LIN {X 0,Y 404.373,Z 885.046,A -85,B 0,C 180,E1 -11042.423,E2 -11042.423} C_VEL
LIN {X 0,Y 404.228,Z 886.16,A -85,B 0,C 180,E1 -11044.238,E2 -11044.238} C_VEL
LIN {X 0,Y 404.158,Z 886.18,A -85,B 0,C 180,E1 -11045.335,E2 -11045.335} C_VEL
LIN {X 0,Y 404.188,Z 885.21,A -85,B 0,C 180,E1 -11047.156,E2 -11047.156} C_VEL
LIN {X 0,Y 404.359,Z 883.5,A -85,B 0,C 180,E1 -11048.595,E2 -11048.595} C_VEL
LIN {X 0,Y 404.64,Z 880.506,A -85,B 0,C 180,E1 -11050.237,E2 -11050.237} C_VEL
LIN {X 0,Y 404.956,Z 876.549,A -85,B 0,C 180,E1 -11051.798,E2 -11051.798} C_VEL
LIN {X 0,Y 405.434,Z 871.294,A -85,B 0,C 180,E1 -11053.382,E2 -11053.382} C_VEL
LIN {X 0,Y 405.955,Z 864.651,A -85,B 0,C 180,E1 -11054.95,E2 -11054.95} C_VEL
LIN {X 0,Y 406.678,Z 856.301,A -85,B 0,C 180,E1 -11056.51,E2 -11056.51} C_VEL
LIN {X 0,Y 407.287,Z 847.808,A -85,B 0,C 180,E1 -11057.798,E2 -11057.798} C_VEL
LIN {X 0,Y 407.94,Z 838.484,A -85,B 0,C 180,E1 -11058.952,E2 -11058.952} C_VEL
LIN {X 0,Y 408.542,Z 828.149,A -85,B 0,C 180,E1 -11059.986,E2 -11059.986} C_VEL
LIN {X 0,Y 409.118,Z 817.223,A -85,B 0,C 180,E1 -11060.858,E2 -11060.858} C_VEL
LIN {X 0,Y 409.51,Z 805.087,A -85,B 0,C 180,E1 -11061.613,E2 -11061.613} C_VEL
LIN {X 0,Y 409.764,Z 792.492,A -85,B 0,C 180,E1 -11062.177,E2 -11062.177} C_VEL
LIN {X 0,Y 409.872,Z 779.499,A -85,B 0,C 180,E1 -11062.551,E2 -11062.551} C_VEL
LIN {X 0,Y 410.43,Z 724.572,A -85,B 0,C 180,E1 -11063.541,E2 -11063.541} C_VEL
LIN {X 0,Y 409.821,Z 721.492,A -85,B 0,C 180,E1 -11063.627,E2 -11063.627} C_VEL
LIN {X 0,Y 407.436,Z 717.769,A -85,B 0,C 180,E1 -11063.81,E2 -11063.81} C_VEL
LIN {X 0,Y 401.011,Z 711.142,A -85,B 0,C 180,E1 -11064.25,E2 -11064.25} C_VEL
LIN {X 0,Y 399.002,Z 707.692,A -85,B 0,C 180,E1 -11064.415,E2 -11064.415} C_VEL
LIN {X 0,Y 397.415,Z 703.698,A -85,B 0,C 180,E1 -11064.614,E2 -11064.614} C_VEL
LIN {X 0,Y 397.262,Z 703.081,A -85,B 0,C 180,E1 -11064.787,E2 -11064.787} C_VEL
LIN {X 0,Y 397.442,Z 702.978,A -85,B 0,C 180,E1 -11067.975,E2 -11067.975} C_VEL
LIN {X 0,Y 397.441,Z 702.977,A -85,B 0,C 180,E1 -11072.028,E2 -11072.028} C_VEL
LIN {X 0,Y 397.324,Z 702.996,A -85,B 0,C 180,E1 -11076.094,E2 -11076.094} C_VEL
LIN {X 0,Y 397.23,Z 703.003,A -85,B 0,C 180,E1 -11079.164,E2 -11079.164} C_VEL
LIN {X 0,Y 397.218,Z 703.004,A -85,B 0,C 180,E1 -11082.26,E2 -11082.26} C_VEL
LIN {X 0,Y 397.178,Z 703.005,A -85,B 0,C 180,E1 -11085.393,E2 -11085.393} C_VEL
LIN {X 0,Y 397.146,Z 703.013,A -85,B 0,C 180,E1 -11088.576,E2 -11088.576} C_VEL
LIN {X 0,Y 397.098,Z 703.016,A -85,B 0,C 180,E1 -11091.82,E2 -11091.82} C_VEL
LIN {X 0,Y 397.107,Z 703.011,A -85,B 0,C 180,E1 -11095.136,E2 -11095.136} C_VEL
LIN {X 0,Y 397.066,Z 703.017,A -85,B 0,C 180,E1 -11098.55,E2 -11098.55} C_VEL
LIN {X 0,Y 397.081,Z 703.017,A -85,B 0,C 180,E1 -11101.835,E2 -11101.835} C_VEL
LIN {X 0,Y 397.121,Z 702.997,A -85,B 0,C 180,E1 -11104.495,E2 -11104.495} C_VEL
LIN {X 0,Y 397.092,Z 703.016,A -85,B 0,C 180,E1 -11108.278,E2 -11108.278} C_VEL
LIN {X 0,Y 397.051,Z 703.024,A -85,B 0,C 180,E1 -11110.915,E2 -11110.915} C_VEL
LIN {X 0,Y 397.083,Z 703.02,A -85,B 0,C 180,E1 -11114.93,E2 -11114.93} C_VEL
LIN {X 0,Y 397.057,Z 703.026,A -85,B 0,C 180,E1 -11118.024,E2 -11118.024} C_VEL
LIN {X 0,Y 397.093,Z 703.02,A -85,B 0,C 180,E1 -11121.147,E2 -11121.147} C_VEL
LIN {X 0,Y 397.096,Z 703.021,A -85,B 0,C 180,E1 -11124.503,E2 -11124.503} C_VEL
LIN {X 0,Y 397.119,Z 703.2,A -85,B 0,C 180,E1 -11127.857,E2 -11127.857} C_VEL
LIN {X 0,Y 397.298,Z 704.02,A -85,B 0,C 180,E1 -11128.009,E2 -11128.009} C_VEL
LIN {X 0,Y 402.683,Z 719.124,A -85,B 0,C 180,E1 -11128.58,E2 -11128.58} C_VEL
LIN {X 0,Y 401.817,Z 779.52,A -85,B 0,C 180,E1 -11129.829,E2 -11129.829} C_VEL
LIN {X 0,Y 401.599,Z 791.294,A -85,B 0,C 180,E1 -11130.227,E2 -11130.227} C_VEL
LIN {X 0,Y 401.342,Z 801.779,A -85,B 0,C 180,E1 -11130.724,E2 -11130.724} C_VEL
LIN {X 0,Y 401.038,Z 811.202,A -85,B 0,C 180,E1 -11131.293,E2 -11131.293} C_VEL
LIN {X 0,Y 400.595,Z 820.808,A -85,B 0,C 180,E1 -11132.011,E2 -11132.011} C_VEL
LIN {X 0,Y 400.075,Z 831.074,A -85,B 0,C 180,E1 -11132.962,E2 -11132.962} C_VEL
LIN {X 0,Y 399.546,Z 839.6,A -85,B 0,C 180,E1 -11133.912,E2 -11133.912} C_VEL
LIN {X 0,Y 399.101,Z 847.754,A -85,B 0,C 180,E1 -11134.999,E2 -11134.999} C_VEL
LIN {X 0,Y 398.681,Z 854.642,A -85,B 0,C 180,E1 -11136.081,E2 -11136.081} C_VEL
LIN {X 0,Y 398.145,Z 861.775,A -85,B 0,C 180,E1 -11137.422,E2 -11137.422} C_VEL
LIN {X 0,Y 397.75,Z 867.648,A -85,B 0,C 180,E1 -11138.763,E2 -11138.763} C_VEL
LIN {X 0,Y 397.539,Z 871.976,A -85,B 0,C 180,E1 -11139.945,E2 -11139.945} C_VEL
LIN {X 0,Y 397.261,Z 876.335,A -85,B 0,C 180,E1 -11141.431,E2 -11141.431} C_VEL
LIN {X 0,Y 397.098,Z 879.609,A -85,B 0,C 180,E1 -11142.888,E2 -11142.888} C_VEL
LIN {X 0,Y 396.942,Z 882.245,A -85,B 0,C 180,E1 -11144.598,E2 -11144.598} C_VEL
LIN {X 0,Y 396.906,Z 883.373,A -85,B 0,C 180,E1 -11145.647,E2 -11145.647} C_VEL
LIN {X 0,Y 396.939,Z 883.999,A -85,B 0,C 180,E1 -11146.861,E2 -11146.861} C_VEL
LIN {X 0,Y 397.061,Z 883.862,A -85,B 0,C 180,E1 -11148.773,E2 -11148.773} C_VEL
LIN {X 0,Y 397.327,Z 881.934,A -85,B 0,C 180,E1 -11150.84,E2 -11150.84} C_VEL
LIN {X 0,Y 397.605,Z 879.747,A -85,B 0,C 180,E1 -11152.211,E2 -11152.211} C_VEL
LIN {X 0,Y 397.873,Z 877.209,A -85,B 0,C 180,E1 -11153.407,E2 -11153.407} C_VEL
LIN {X 0,Y 398.275,Z 872.869,A -85,B 0,C 180,E1 -11154.938,E2 -11154.938} C_VEL
LIN {X 0,Y 398.75,Z 867.283,A -85,B 0,C 180,E1 -11156.463,E2 -11156.463} C_VEL
LIN {X 0,Y 399.295,Z 861.568,A -85,B 0,C 180,E1 -11157.73,E2 -11157.73} C_VEL
LIN {X 0,Y 399.927,Z 854.651,A -85,B 0,C 180,E1 -11158.993,E2 -11158.993} C_VEL
LIN {X 0,Y 400.608,Z 846.07,A -85,B 0,C 180,E1 -11160.276,E2 -11160.276} C_VEL
LIN {X 0,Y 401.152,Z 838.689,A -85,B 0,C 180,E1 -11161.2,E2 -11161.2} C_VEL
LIN {X 0,Y 401.806,Z 829.752,A -85,B 0,C 180,E1 -11162.13,E2 -11162.13} C_VEL
LIN {X 0,Y 402.229,Z 821.185,A -85,B 0,C 180,E1 -11162.879,E2 -11162.879} C_VEL
LIN {X 0,Y 402.653,Z 810.512,A -85,B 0,C 180,E1 -11163.627,E2 -11163.627} C_VEL
LIN {X 0,Y 403.032,Z 800.219,A -85,B 0,C 180,E1 -11164.187,E2 -11164.187} C_VEL
LIN {X 0,Y 403.228,Z 789.583,A -85,B 0,C 180,E1 -11164.624,E2 -11164.624} C_VEL
LIN {X 0,Y 403.267,Z 777.527,A -85,B 0,C 180,E1 -11164.968,E2 -11164.968} C_VEL
LIN {X 0,Y 404.446,Z 720.258,A -85,B 0,C 180,E1 -11166.218,E2 -11166.218} C_VEL
LIN {X 0,Y 399.902,Z 709.007,A -85,B 0,C 180,E1 -11166.793,E2 -11166.793} C_VEL
LIN {X 0,Y 397.46,Z 703.744,A -85,B 0,C 180,E1 -11167.138,E2 -11167.138} C_VEL
LIN {X 0,Y 397.343,Z 703.058,A -85,B 0,C 180,E1 -11167.339,E2 -11167.339} C_VEL
LIN {X 0,Y 397.205,Z 703.008,A -85,B 0,C 180,E1 -11171.223,E2 -11171.223} C_VEL
LIN {X 0,Y 397.184,Z 703.011,A -85,B 0,C 180,E1 -11174.343,E2 -11174.343} C_VEL
LIN {X 0,Y 397.152,Z 703.013,A -85,B 0,C 180,E1 -11177.508,E2 -11177.508} C_VEL
LIN {X 0,Y 397.11,Z 703.021,A -85,B 0,C 180,E1 -11180.729,E2 -11180.729} C_VEL
LIN {X 0,Y 397.131,Z 703.015,A -85,B 0,C 180,E1 -11184.018,E2 -11184.018} C_VEL
LIN {X 0,Y 397.122,Z 703.017,A -85,B 0,C 180,E1 -11187.763,E2 -11187.763} C_VEL
LIN {X 0,Y 397.085,Z 703.023,A -85,B 0,C 180,E1 -11190.882,E2 -11190.882} C_VEL
LIN {X 0,Y 397.131,Z 703.015,A -85,B 0,C 180,E1 -11194.493,E2 -11194.493} C_VEL
LIN {X 0,Y 397.11,Z 703.018,A -85,B 0,C 180,E1 -11198.274,E2 -11198.274} C_VEL
LIN {X 0,Y 397.095,Z 703.021,A -85,B 0,C 180,E1 -11200.908,E2 -11200.908} C_VEL
LIN {X 0,Y 397.108,Z 703.021,A -85,B 0,C 180,E1 -11203.648,E2 -11203.648} C_VEL
LIN {X 0,Y 397.108,Z 703.018,A -85,B 0,C 180,E1 -11206.52,E2 -11206.52} C_VEL
LIN {X 0,Y 397.118,Z 703.016,A -85,B 0,C 180,E1 -11210.422,E2 -11210.422} C_VEL
LIN {X 0,Y 397.113,Z 703.018,A -85,B 0,C 180,E1 -11214.264,E2 -11214.264} C_VEL
LIN {X 0,Y 397.152,Z 703.193,A -85,B 0,C 180,E1 -11216.375,E2 -11216.375} C_VEL
LIN {X 0,Y 401.047,Z 719.548,A -85,B 0,C 180,E1 -11219.455,E2 -11219.455} C_VEL
LIN {X 0,Y 402.871,Z 729.169,A -85,B 0,C 180,E1 -11221.156,E2 -11221.156} C_VEL
LIN {X 0,Y 400.963,Z 752.371,A -85,B 0,C 180,E1 -11224.845,E2 -11224.845} C_VEL
LIN {X 0,Y 399.627,Z 772.769,A -85,B 0,C 180,E1 -11228.054,E2 -11228.054} C_VEL
LIN {X 0,Y 398.971,Z 784.14,A -85,B 0,C 180,E1 -11229.808,E2 -11229.808} C_VEL
LIN {X 0,Y 400.351,Z 797.906,A -85,B 0,C 180,E1 -11230.261,E2 -11230.261} C_VEL
LIN {X 0,Y 403.016,Z 825.383,A -85,B 0,C 180,E1 -11230.899,E2 -11230.899} C_VEL
LIN {X 0,Y 402.062,Z 895.502,A -85,B 0,C 180,E1 -11232.186,E2 -11232.186} C_VEL
LIN {X 0,Y 401.522,Z 908.77,A -85,B 0,C 180,E1 -11232.622,E2 -11232.622} C_VEL
LIN {X 0,Y 400.721,Z 921.535,A -85,B 0,C 180,E1 -11233.243,E2 -11233.243} C_VEL
LIN {X 0,Y 399.835,Z 933.73,A -85,B 0,C 180,E1 -11234.058,E2 -11234.058} C_VEL
LIN {X 0,Y 398.861,Z 945.354,A -85,B 0,C 180,E1 -11235.065,E2 -11235.065} C_VEL
LIN {X 0,Y 398.127,Z 955.313,A -85,B 0,C 180,E1 -11236.144,E2 -11236.144} C_VEL
LIN {X 0,Y 397.63,Z 963.618,A -85,B 0,C 180,E1 -11237.235,E2 -11237.235} C_VEL
LIN {X 0,Y 397.003,Z 971.74,A -85,B 0,C 180,E1 -11238.511,E2 -11238.511} C_VEL
LIN {X 0,Y 396.572,Z 979.734,A -85,B 0,C 180,E1 -11240.049,E2 -11240.049} C_VEL
LIN {X 0,Y 396.359,Z 987.083,A -85,B 0,C 180,E1 -11241.844,E2 -11241.844} C_VEL
LIN {X 0,Y 396.291,Z 991.709,A -85,B 0,C 180,E1 -11243.281,E2 -11243.281} C_VEL
LIN {X 0,Y 396.396,Z 995.766,A -85,B 0,C 180,E1 -11244.913,E2 -11244.913} C_VEL
LIN {X 0,Y 396.519,Z 997.717,A -85,B 0,C 180,E1 -11245.933,E2 -11245.933} C_VEL
LIN {X 0,Y 396.457,Z 999.165,A -85,B 0,C 180,E1 -11246.95,E2 -11246.95} C_VEL
LIN {X 0,Y 396.478,Z 1000.191,A -85,B 0,C 180,E1 -11247.967,E2 -11247.967} C_VEL
LIN {X 0,Y 396.511,Z 1000.812,A -85,B 0,C 180,E1 -11248.983,E2 -11248.983} C_VEL
LIN {X 0,Y 396.541,Z 1001.028,A -85,B 0,C 180,E1 -11249.998,E2 -11249.998} C_VEL
LIN {X 0,Y 396.513,Z 1000.791,A -85,B 0,C 180,E1 -11251.014,E2 -11251.014} C_VEL
LIN {X 0,Y 396.483,Z 1000.134,A -85,B 0,C 180,E1 -11252.03,E2 -11252.03} C_VEL
LIN {X 0,Y 396.461,Z 999.074,A -85,B 0,C 180,E1 -11253.047,E2 -11253.047} C_VEL
LIN {X 0,Y 396.504,Z 997.609,A -85,B 0,C 180,E1 -11254.064,E2 -11254.064} C_VEL
LIN {X 0,Y 396.319,Z 994.499,A -85,B 0,C 180,E1 -11255.596,E2 -11255.596} C_VEL
LIN {X 0,Y 396.307,Z 990.341,A -85,B 0,C 180,E1 -11257.129,E2 -11257.129} C_VEL
LIN {X 0,Y 396.413,Z 983.991,A -85,B 0,C 180,E1 -11258.923,E2 -11258.923} C_VEL
LIN {X 0,Y 396.648,Z 977.08,A -85,B 0,C 180,E1 -11260.462,E2 -11260.462} C_VEL
LIN {X 0,Y 397.159,Z 968.562,A -85,B 0,C 180,E1 -11261.999,E2 -11261.999} C_VEL
LIN {X 0,Y 397.892,Z 959.904,A -85,B 0,C 180,E1 -11263.273,E2 -11263.273} C_VEL
LIN {X 0,Y 398.548,Z 950.429,A -85,B 0,C 180,E1 -11264.421,E2 -11264.421} C_VEL
LIN {X 0,Y 399.276,Z 940.172,A -85,B 0,C 180,E1 -11265.438,E2 -11265.438} C_VEL
LIN {X 0,Y 400.222,Z 929.079,A -85,B 0,C 180,E1 -11266.316,E2 -11266.316} C_VEL
LIN {X 0,Y 401.113,Z 916.855,A -85,B 0,C 180,E1 -11267.065,E2 -11267.065} C_VEL
LIN {X 0,Y 401.862,Z 904.313,A -85,B 0,C 180,E1 -11267.622,E2 -11267.622} C_VEL
LIN {X 0,Y 402.353,Z 891.365,A -85,B 0,C 180,E1 -11267.994,E2 -11267.994} C_VEL
LIN {X 0,Y 403.171,Z 822.843,A -85,B 0,C 180,E1 -11269.249,E2 -11269.249} C_VEL
LIN {X 0,Y 399.24,Z 786.031,A -85,B 0,C 180,E1 -11270.158,E2 -11270.158} C_VEL
LIN {X 0,Y 398.849,Z 782.941,A -85,B 0,C 180,E1 -11270.263,E2 -11270.263} C_VEL
LIN {X 0,Y 400.24,Z 761.86,A -85,B 0,C 180,E1 -11273.544,E2 -11273.544} C_VEL
LIN {X 0,Y 402.273,Z 734.827,A -85,B 0,C 180,E1 -11277.86,E2 -11277.86} C_VEL
LIN {X 0,Y 402.746,Z 727.843,A -85,B 0,C 180,E1 -11278.999,E2 -11278.999} C_VEL
LIN {X 0,Y 400.176,Z 715.833,A -85,B 0,C 180,E1 -11281.201,E2 -11281.201} C_VEL
LIN {X 0,Y 397.136,Z 703.138,A -85,B 0,C 180,E1 -11283.696,E2 -11283.696} C_VEL
LIN {X 0,Y 397.087,Z 703.023,A -85,B 0,C 180,E1 -11287.207,E2 -11287.207} C_VEL
LIN {X 0,Y 397.094,Z 703.019,A -85,B 0,C 180,E1 -11290.444,E2 -11290.444} C_VEL
LIN {X 0,Y 397.093,Z 703.018,A -85,B 0,C 180,E1 -11293.647,E2 -11293.647} C_VEL
LIN {X 0,Y 397.097,Z 703.015,A -85,B 0,C 180,E1 -11296.519,E2 -11296.519} C_VEL
LIN {X 0,Y 397.105,Z 703.009,A -85,B 0,C 180,E1 -11300.422,E2 -11300.422} C_VEL
LIN {X 0,Y 397.099,Z 703.01,A -85,B 0,C 180,E1 -11304.264,E2 -11304.264} C_VEL
LIN {X 0,Y 397.104,Z 703.018,A -85,B 0,C 180,E1 -11306.726,E2 -11306.726} C_VEL
LIN {X 0,Y 397.123,Z 703.016,A -85,B 0,C 180,E1 -11310.296,E2 -11310.296} C_VEL
LIN {X 0,Y 397.184,Z 703.006,A -85,B 0,C 180,E1 -11312.609,E2 -11312.609} C_VEL
LIN {X 0,Y 397.122,Z 703.017,A -85,B 0,C 180,E1 -11315.981,E2 -11315.981} C_VEL
LIN {X 0,Y 397.127,Z 703.016,A -85,B 0,C 180,E1 -11319.704,E2 -11319.704} C_VEL
LIN {X 0,Y 397.172,Z 703.002,A -85,B 0,C 180,E1 -11322.843,E2 -11322.843} C_VEL
LIN {X 0,Y 397.166,Z 703.012,A -85,B 0,C 180,E1 -11325.657,E2 -11325.657} C_VEL
LIN {X 0,Y 397.187,Z 703.007,A -85,B 0,C 180,E1 -11328.776,E2 -11328.776} C_VEL
LIN {X 0,Y 397.349,Z 702.985,A -85,B 0,C 180,E1 -11332.076,E2 -11332.076} C_VEL
LIN {X 0,Y 397.243,Z 702.996,A -85,B 0,C 180,E1 -11334.925,E2 -11334.925} C_VEL
LIN {X 0,Y 397.44,Z 702.977,A -85,B 0,C 180,E1 -11337.973,E2 -11337.973} C_VEL
LIN {X 0,Y 397.568,Z 702.957,A -85,B 0,C 180,E1 -11340,E2 -11340} C_VEL
LIN {X 0,Y 397.369,Z 702.983,A -85,B 0,C 180,E1 -11343.042,E2 -11343.042} C_VEL
LIN {X 0,Y 397.35,Z 702.987,A -85,B 0,C 180,E1 -11347.112,E2 -11347.112} C_VEL
LIN {X 0,Y 397.207,Z 703.005,A -85,B 0,C 180,E1 -11350.192,E2 -11350.192} C_VEL
LIN {X 0,Y 397.215,Z 703.005,A -85,B 0,C 180,E1 -11353.322,E2 -11353.322} C_VEL
LIN {X 0,Y 397.17,Z 703.014,A -85,B 0,C 180,E1 -11357.156,E2 -11357.156} C_VEL
LIN {X 0,Y 397.091,Z 703.021,A -85,B 0,C 180,E1 -11360.731,E2 -11360.731} C_VEL
LIN {X 0,Y 397.114,Z 703.006,A -85,B 0,C 180,E1 -11364.02,E2 -11364.02} C_VEL
LIN {X 0,Y 397.184,Z 703.006,A -85,B 0,C 180,E1 -11367.391,E2 -11367.391} C_VEL
LIN {X 0,Y 397.069,Z 703.026,A -85,B 0,C 180,E1 -11370.884,E2 -11370.884} C_VEL
LIN {X 0,Y 397.117,Z 703.017,A -85,B 0,C 180,E1 -11374.495,E2 -11374.495} C_VEL
LIN {X 0,Y 397.099,Z 703.016,A -85,B 0,C 180,E1 -11378.276,E2 -11378.276} C_VEL
LIN {X 0,Y 397.082,Z 703.02,A -85,B 0,C 180,E1 -11380.91,E2 -11380.91} C_VEL
LIN {X 0,Y 397.094,Z 703.022,A -85,B 0,C 180,E1 -11383.65,E2 -11383.65} C_VEL
LIN {X 0,Y 397.133,Z 703.284,A -85,B 0,C 180,E1 -11385.063,E2 -11385.063} C_VEL
LIN {X 0,Y 397.457,Z 704.485,A -85,B 0,C 180,E1 -11385.222,E2 -11385.222} C_VEL
LIN {X 0,Y 404.151,Z 720.562,A -85,B 0,C 180,E1 -11385.923,E2 -11385.923} C_VEL
LIN {X 0,Y 403.609,Z 785.345,A -85,B 0,C 180,E1 -11387.147,E2 -11387.147} C_VEL
LIN {X 0,Y 403.48,Z 798.403,A -85,B 0,C 180,E1 -11387.593,E2 -11387.593} C_VEL
LIN {X 0,Y 403.24,Z 810.296,A -85,B 0,C 180,E1 -11388.193,E2 -11388.193} C_VEL
LIN {X 0,Y 402.814,Z 821.878,A -85,B 0,C 180,E1 -11388.972,E2 -11388.972} C_VEL
LIN {X 0,Y 402.139,Z 832.712,A -85,B 0,C 180,E1 -11389.906,E2 -11389.906} C_VEL
LIN {X 0,Y 401.408,Z 843.546,A -85,B 0,C 180,E1 -11391.091,E2 -11391.091} C_VEL
LIN {X 0,Y 400.549,Z 853.417,A -85,B 0,C 180,E1 -11392.433,E2 -11392.433} C_VEL
LIN {X 0,Y 399.847,Z 861.013,A -85,B 0,C 180,E1 -11393.711,E2 -11393.711} C_VEL
LIN {X 0,Y 399.259,Z 867.779,A -85,B 0,C 180,E1 -11395.106,E2 -11395.106} C_VEL
LIN {X 0,Y 398.531,Z 874.56,A -85,B 0,C 180,E1 -11396.863,E2 -11396.863} C_VEL
LIN {X 0,Y 397.997,Z 879.692,A -85,B 0,C 180,E1 -11398.608,E2 -11398.608} C_VEL
LIN {X 0,Y 397.636,Z 883.349,A -85,B 0,C 180,E1 -11400.34,E2 -11400.34} C_VEL
LIN {X 0,Y 397.368,Z 885.865,A -85,B 0,C 180,E1 -11402.169,E2 -11402.169} C_VEL
LIN {X 0,Y 397.22,Z 886.998,A -85,B 0,C 180,E1 -11403.75,E2 -11403.75} C_VEL
LIN {X 0,Y 397.17,Z 887.244,A -85,B 0,C 180,E1 -11404.871,E2 -11404.871} C_VEL
LIN {X 0,Y 397.122,Z 887.004,A -85,B 0,C 180,E1 -11405.983,E2 -11405.983} C_VEL
LIN {X 0,Y 397.176,Z 886.288,A -85,B 0,C 180,E1 -11407.092,E2 -11407.092} C_VEL
LIN {X 0,Y 397.304,Z 885.138,A -85,B 0,C 180,E1 -11408.195,E2 -11408.195} C_VEL
LIN {X 0,Y 397.516,Z 883.004,A -85,B 0,C 180,E1 -11409.56,E2 -11409.56} C_VEL
LIN {X 0,Y 397.886,Z 878.772,A -85,B 0,C 180,E1 -11411.463,E2 -11411.463} C_VEL
LIN {X 0,Y 398.337,Z 873.834,A -85,B 0,C 180,E1 -11413.077,E2 -11413.077} C_VEL
LIN {X 0,Y 398.884,Z 867.576,A -85,B 0,C 180,E1 -11414.677,E2 -11414.677} C_VEL
LIN {X 0,Y 399.547,Z 859.778,A -85,B 0,C 180,E1 -11416.265,E2 -11416.265} C_VEL
LIN {X 0,Y 400.195,Z 851.76,A -85,B 0,C 180,E1 -11417.579,E2 -11417.579} C_VEL
LIN {X 0,Y 400.905,Z 841.957,A -85,B 0,C 180,E1 -11418.883,E2 -11418.883} C_VEL
LIN {X 0,Y 401.613,Z 831.064,A -85,B 0,C 180,E1 -11420.051,E2 -11420.051} C_VEL
LIN {X 0,Y 402.227,Z 820.431,A -85,B 0,C 180,E1 -11420.954,E2 -11420.954} C_VEL
LIN {X 0,Y 402.718,Z 807.73,A -85,B 0,C 180,E1 -11421.787,E2 -11421.787} C_VEL
LIN {X 0,Y 403.012,Z 795.141,A -85,B 0,C 180,E1 -11422.392,E2 -11422.392} C_VEL
LIN {X 0,Y 403.092,Z 782.076,A -85,B 0,C 180,E1 -11422.803,E2 -11422.803} C_VEL
LIN {X 0,Y 403.757,Z 720.112,A -85,B 0,C 180,E1 -11423.944,E2 -11423.944} C_VEL
LIN {X 0,Y 399.002,Z 707.692,A -85,B 0,C 180,E1 -11424.415,E2 -11424.415} C_VEL
LIN {X 0,Y 397.975,Z 705.732,A -85,B 0,C 180,E1 -11424.588,E2 -11424.588} C_VEL
LIN {X 0,Y 396.428,Z 704.172,A -85,B 0,C 180,E1 -11424.976,E2 -11424.976} C_VEL
LIN {X 0,Y 394.554,Z 703.476,A -85,B 0,C 180,E1 -11425.595,E2 -11425.595} C_VEL
LIN {X 0,Y 392.119,Z 703.641,A -85,B 0,C 180,E1 -11426.765,E2 -11426.765} C_VEL
LIN {X 0,Y 390.564,Z 703.835,A -85,B 0,C 180,E1 -11428.074,E2 -11428.074} C_VEL
LIN {X 0,Y 390.307,Z 703.866,A -85,B 0,C 180,E1 -11428.738,E2 -11428.738} C_VEL
LIN {X 0,Y 390.407,Z 703.853,A -85,B 0,C 180,E1 -11432.065,E2 -11432.065} C_VEL
LIN {X 0,Y 390.28,Z 703.873,A -85,B 0,C 180,E1 -11436.204,E2 -11436.204} C_VEL
LIN {X 0,Y 390.189,Z 703.879,A -85,B 0,C 180,E1 -11439.331,E2 -11439.331} C_VEL
LIN {X 0,Y 390.201,Z 703.876,A -85,B 0,C 180,E1 -11443.44,E2 -11443.44} C_VEL
LIN {X 0,Y 390.135,Z 703.887,A -85,B 0,C 180,E1 -11447.299,E2 -11447.299} C_VEL
LIN {X 0,Y 390.056,Z 703.892,A -85,B 0,C 180,E1 -11451.124,E2 -11451.124} C_VEL
LIN {X 0,Y 390.048,Z 703.897,A -85,B 0,C 180,E1 -11454.484,E2 -11454.484} C_VEL
LIN {X 0,Y 390.022,Z 703.893,A -85,B 0,C 180,E1 -11457.998,E2 -11457.998} C_VEL
LIN {X 0,Y 390.023,Z 703.899,A -85,B 0,C 180,E1 -11461.506,E2 -11461.506} C_VEL
LIN {X 0,Y 390.073,Z 703.874,A -85,B 0,C 180,E1 -11465.21,E2 -11465.21} C_VEL
LIN {X 0,Y 390.06,Z 703.895,A -85,B 0,C 180,E1 -11469.098,E2 -11469.098} C_VEL
LIN {X 0,Y 390.014,Z 703.9,A -85,B 0,C 180,E1 -11472.369,E2 -11472.369} C_VEL
LIN {X 0,Y 390.049,Z 703.898,A -85,B 0,C 180,E1 -11476.117,E2 -11476.117} C_VEL
LIN {X 0,Y 390.016,Z 703.905,A -85,B 0,C 180,E1 -11479.555,E2 -11479.555} C_VEL
LIN {X 0,Y 390.04,Z 703.899,A -85,B 0,C 180,E1 -11482.452,E2 -11482.452} C_VEL
LIN {X 0,Y 390.069,Z 703.898,A -85,B 0,C 180,E1 -11486.045,E2 -11486.045} C_VEL
LIN {X 0,Y 390.123,Z 704.128,A -85,B 0,C 180,E1 -11487.592,E2 -11487.592} C_VEL
LIN {X 0,Y 390.358,Z 705.253,A -85,B 0,C 180,E1 -11487.748,E2 -11487.748} C_VEL
LIN {X 0,Y 395.91,Z 721.269,A -85,B 0,C 180,E1 -11488.346,E2 -11488.346} C_VEL
LIN {X 0,Y 394.962,Z 779.958,A -85,B 0,C 180,E1 -11489.582,E2 -11489.582} C_VEL
LIN {X 0,Y 394.729,Z 792.276,A -85,B 0,C 180,E1 -11490.005,E2 -11490.005} C_VEL
LIN {X 0,Y 394.45,Z 802.952,A -85,B 0,C 180,E1 -11490.522,E2 -11490.522} C_VEL
LIN {X 0,Y 394.132,Z 812.311,A -85,B 0,C 180,E1 -11491.1,E2 -11491.1} C_VEL
LIN {X 0,Y 393.625,Z 822.748,A -85,B 0,C 180,E1 -11491.906,E2 -11491.906} C_VEL
LIN {X 0,Y 393.176,Z 831.598,A -85,B 0,C 180,E1 -11492.739,E2 -11492.739} C_VEL
LIN {X 0,Y 392.667,Z 839.47,A -85,B 0,C 180,E1 -11493.61,E2 -11493.61} C_VEL
LIN {X 0,Y 392.182,Z 848.423,A -85,B 0,C 180,E1 -11494.811,E2 -11494.811} C_VEL
LIN {X 0,Y 391.686,Z 855.962,A -85,B 0,C 180,E1 -11496.018,E2 -11496.018} C_VEL
LIN {X 0,Y 391.176,Z 862.568,A -85,B 0,C 180,E1 -11497.277,E2 -11497.277} C_VEL
LIN {X 0,Y 390.769,Z 868.495,A -85,B 0,C 180,E1 -11498.642,E2 -11498.642} C_VEL
LIN {X 0,Y 390.506,Z 873.35,A -85,B 0,C 180,E1 -11500.004,E2 -11500.004} C_VEL
LIN {X 0,Y 390.322,Z 876.62,A -85,B 0,C 180,E1 -11501.089,E2 -11501.089} C_VEL
LIN {X 0,Y 390.105,Z 880.376,A -85,B 0,C 180,E1 -11502.717,E2 -11502.717} C_VEL
LIN {X 0,Y 389.942,Z 882.979,A -85,B 0,C 180,E1 -11504.315,E2 -11504.315} C_VEL
LIN {X 0,Y 389.926,Z 884.907,A -85,B 0,C 180,E1 -11506.449,E2 -11506.449} C_VEL
LIN {X 0,Y 389.973,Z 885.178,A -85,B 0,C 180,E1 -11507.51,E2 -11507.51} C_VEL
LIN {X 0,Y 390.045,Z 885.029,A -85,B 0,C 180,E1 -11508.568,E2 -11508.568} C_VEL
LIN {X 0,Y 390.318,Z 883.425,A -85,B 0,C 180,E1 -11510.674,E2 -11510.674} C_VEL
LIN {X 0,Y 390.551,Z 881.871,A -85,B 0,C 180,E1 -11511.789,E2 -11511.789} C_VEL
LIN {X 0,Y 391.002,Z 877.693,A -85,B 0,C 180,E1 -11513.809,E2 -11513.809} C_VEL
LIN {X 0,Y 391.44,Z 873.179,A -85,B 0,C 180,E1 -11515.366,E2 -11515.366} C_VEL
LIN {X 0,Y 391.893,Z 868.496,A -85,B 0,C 180,E1 -11516.659,E2 -11516.659} C_VEL
LIN {X 0,Y 392.474,Z 862.791,A -85,B 0,C 180,E1 -11517.947,E2 -11517.947} C_VEL
LIN {X 0,Y 393.152,Z 855.878,A -85,B 0,C 180,E1 -11519.232,E2 -11519.232} C_VEL
LIN {X 0,Y 393.791,Z 848.202,A -85,B 0,C 180,E1 -11520.416,E2 -11520.416} C_VEL
LIN {X 0,Y 394.408,Z 840.397,A -85,B 0,C 180,E1 -11521.426,E2 -11521.426} C_VEL
LIN {X 0,Y 395.143,Z 831.072,A -85,B 0,C 180,E1 -11522.421,E2 -11522.421} C_VEL
LIN {X 0,Y 395.589,Z 822.591,A -85,B 0,C 180,E1 -11523.182,E2 -11523.182} C_VEL
LIN {X 0,Y 396.04,Z 812.049,A -85,B 0,C 180,E1 -11523.943,E2 -11523.943} C_VEL
LIN {X 0,Y 396.451,Z 801.233,A -85,B 0,C 180,E1 -11524.544,E2 -11524.544} C_VEL
LIN {X 0,Y 396.662,Z 791.48,A -85,B 0,C 180,E1 -11524.955,E2 -11524.955} C_VEL
LIN {X 0,Y 396.704,Z 779.594,A -85,B 0,C 180,E1 -11525.31,E2 -11525.31} C_VEL
LIN {X 0,Y 397.972,Z 722.063,A -85,B 0,C 180,E1 -11526.603,E2 -11526.603} C_VEL
LIN {X 0,Y 393.994,Z 712.253,A -85,B 0,C 180,E1 -11527.134,E2 -11527.134} C_VEL
LIN {X 0,Y 390.503,Z 704.876,A -85,B 0,C 180,E1 -11527.612,E2 -11527.612} C_VEL
LIN {X 0,Y 390.301,Z 704.011,A -85,B 0,C 180,E1 -11527.799,E2 -11527.799} C_VEL
LIN {X 0,Y 390.154,Z 703.885,A -85,B 0,C 180,E1 -11531.429,E2 -11531.429} C_VEL
LIN {X 0,Y 390.151,Z 703.889,A -85,B 0,C 180,E1 -11534.607,E2 -11534.607} C_VEL
LIN {X 0,Y 390.119,Z 703.89,A -85,B 0,C 180,E1 -11537.834,E2 -11537.834} C_VEL
LIN {X 0,Y 390.063,Z 703.897,A -85,B 0,C 180,E1 -11541.122,E2 -11541.122} C_VEL
LIN {X 0,Y 390.068,Z 703.899,A -85,B 0,C 180,E1 -11544.481,E2 -11544.481} C_VEL
LIN {X 0,Y 390.077,Z 703.895,A -85,B 0,C 180,E1 -11548.012,E2 -11548.012} C_VEL
LIN {X 0,Y 390.03,Z 703.901,A -85,B 0,C 180,E1 -11551.504,E2 -11551.504} C_VEL
LIN {X 0,Y 390.091,Z 703.895,A -85,B 0,C 180,E1 -11555.206,E2 -11555.206} C_VEL
LIN {X 0,Y 390.077,Z 703.895,A -85,B 0,C 180,E1 -11559.218,E2 -11559.218} C_VEL
LIN {X 0,Y 390.049,Z 703.898,A -85,B 0,C 180,E1 -11562.373,E2 -11562.373} C_VEL
LIN {X 0,Y 390.05,Z 703.899,A -85,B 0,C 180,E1 -11565.354,E2 -11565.354} C_VEL
LIN {X 0,Y 390.037,Z 703.899,A -85,B 0,C 180,E1 -11568.186,E2 -11568.186} C_VEL
LIN {X 0,Y 390.092,Z 703.891,A -85,B 0,C 180,E1 -11570.906,E2 -11570.906} C_VEL
LIN {X 0,Y 390.09,Z 703.895,A -85,B 0,C 180,E1 -11574.792,E2 -11574.792} C_VEL
LIN {X 0,Y 390.107,Z 704.11,A -85,B 0,C 180,E1 -11576.048,E2 -11576.048} C_VEL
LIN {X 0,Y 393.989,Z 720.426,A -85,B 0,C 180,E1 -11579.178,E2 -11579.178} C_VEL
LIN {X 0,Y 395.966,Z 729.865,A -85,B 0,C 180,E1 -11580.895,E2 -11580.895} C_VEL
LIN {X 0,Y 394.314,Z 749.65,A -85,B 0,C 180,E1 -11584.107,E2 -11584.107} C_VEL
LIN {X 0,Y 392.947,Z 768.33,A -85,B 0,C 180,E1 -11587.106,E2 -11587.106} C_VEL
LIN {X 0,Y 392.06,Z 782.688,A -85,B 0,C 180,E1 -11589.35,E2 -11589.35} C_VEL
LIN {X 0,Y 393.846,Z 799.08,A -85,B 0,C 180,E1 -11589.891,E2 -11589.891} C_VEL
LIN {X 0,Y 395.737,Z 819.145,A -85,B 0,C 180,E1 -11590.45,E2 -11590.45} C_VEL
LIN {X 0,Y 396.249,Z 826.893,A -85,B 0,C 180,E1 -11590.621,E2 -11590.621} C_VEL
LIN {X 0,Y 395.237,Z 895.17,A -85,B 0,C 180,E1 -11591.902,E2 -11591.902} C_VEL
LIN {X 0,Y 394.697,Z 908.22,A -85,B 0,C 180,E1 -11592.345,E2 -11592.345} C_VEL
LIN {X 0,Y 393.808,Z 921.412,A -85,B 0,C 180,E1 -11593.007,E2 -11593.007} C_VEL
LIN {X 0,Y 392.844,Z 934.16,A -85,B 0,C 180,E1 -11593.9,E2 -11593.9} C_VEL
LIN {X 0,Y 391.843,Z 945.524,A -85,B 0,C 180,E1 -11594.924,E2 -11594.924} C_VEL
LIN {X 0,Y 391.064,Z 955.423,A -85,B 0,C 180,E1 -11596.039,E2 -11596.039} C_VEL
LIN {X 0,Y 390.473,Z 964.289,A -85,B 0,C 180,E1 -11597.261,E2 -11597.261} C_VEL
LIN {X 0,Y 389.811,Z 973.507,A -85,B 0,C 180,E1 -11598.823,E2 -11598.823} C_VEL
LIN {X 0,Y 389.432,Z 980.964,A -85,B 0,C 180,E1 -11600.389,E2 -11600.389} C_VEL
LIN {X 0,Y 389.301,Z 986.03,A -85,B 0,C 180,E1 -11601.695,E2 -11601.695} C_VEL
LIN {X 0,Y 389.237,Z 990.936,A -85,B 0,C 180,E1 -11603.253,E2 -11603.253} C_VEL
LIN {X 0,Y 389.315,Z 994.73,A -85,B 0,C 180,E1 -11604.82,E2 -11604.82} C_VEL
LIN {X 0,Y 389.462,Z 996.69,A -85,B 0,C 180,E1 -11605.859,E2 -11605.859} C_VEL
LIN {X 0,Y 389.418,Z 998.147,A -85,B 0,C 180,E1 -11606.895,E2 -11606.895} C_VEL
LIN {X 0,Y 389.44,Z 999.176,A -85,B 0,C 180,E1 -11607.93,E2 -11607.93} C_VEL
LIN {X 0,Y 389.478,Z 999.8,A -85,B 0,C 180,E1 -11608.965,E2 -11608.965} C_VEL
LIN {X 0,Y 389.513,Z 1000.019,A -85,B 0,C 180,E1 -11609.998,E2 -11609.998} C_VEL
LIN {X 0,Y 389.48,Z 999.786,A -85,B 0,C 180,E1 -11611.032,E2 -11611.032} C_VEL
LIN {X 0,Y 389.444,Z 999.129,A -85,B 0,C 180,E1 -11612.067,E2 -11612.067} C_VEL
LIN {X 0,Y 389.418,Z 998.068,A -85,B 0,C 180,E1 -11613.102,E2 -11613.102} C_VEL
LIN {X 0,Y 389.45,Z 996.602,A -85,B 0,C 180,E1 -11614.138,E2 -11614.138} C_VEL
LIN {X 0,Y 389.253,Z 993.49,A -85,B 0,C 180,E1 -11615.697,E2 -11615.697} C_VEL
LIN {X 0,Y 389.236,Z 989.332,A -85,B 0,C 180,E1 -11617.259,E2 -11617.259} C_VEL
LIN {X 0,Y 389.346,Z 982.985,A -85,B 0,C 180,E1 -11619.086,E2 -11619.086} C_VEL
LIN {X 0,Y 389.623,Z 976.078,A -85,B 0,C 180,E1 -11620.653,E2 -11620.653} C_VEL
LIN {X 0,Y 390.117,Z 967.558,A -85,B 0,C 180,E1 -11622.219,E2 -11622.219} C_VEL
LIN {X 0,Y 390.855,Z 958.91,A -85,B 0,C 180,E1 -11623.517,E2 -11623.517} C_VEL
LIN {X 0,Y 391.667,Z 948.269,A -85,B 0,C 180,E1 -11624.813,E2 -11624.813} C_VEL
LIN {X 0,Y 392.562,Z 937.808,A -85,B 0,C 180,E1 -11625.842,E2 -11625.842} C_VEL
LIN {X 0,Y 393.542,Z 926.418,A -85,B 0,C 180,E1 -11626.734,E2 -11626.734} C_VEL
LIN {X 0,Y 394.41,Z 914.901,A -85,B 0,C 180,E1 -11627.431,E2 -11627.431} C_VEL
LIN {X 0,Y 395.192,Z 901.83,A -85,B 0,C 180,E1 -11627.997,E2 -11627.997} C_VEL
LIN {X 0,Y 395.677,Z 887.99,A -85,B 0,C 180,E1 -11628.376,E2 -11628.376} C_VEL
LIN {X 0,Y 396.498,Z 823.718,A -85,B 0,C 180,E1 -11629.566,E2 -11629.566} C_VEL
LIN {X 0,Y 392.532,Z 786.738,A -85,B 0,C 180,E1 -11630.5,E2 -11630.5} C_VEL
LIN {X 0,Y 391.944,Z 781.723,A -85,B 0,C 180,E1 -11630.67,E2 -11630.67} C_VEL
LIN {X 0,Y 393.55,Z 759.25,A -85,B 0,C 180,E1 -11634.249,E2 -11634.249} C_VEL
LIN {X 0,Y 395.416,Z 735.659,A -85,B 0,C 180,E1 -11638.097,E2 -11638.097} C_VEL
LIN {X 0,Y 395.884,Z 729.647,A -85,B 0,C 180,E1 -11639.094,E2 -11639.094} C_VEL
LIN {X 0,Y 393.106,Z 716.682,A -85,B 0,C 180,E1 -11641.527,E2 -11641.527} C_VEL
LIN {X 0,Y 390.099,Z 704.003,A -85,B 0,C 180,E1 -11644.089,E2 -11644.089} C_VEL
LIN {X 0,Y 390.036,Z 703.9,A -85,B 0,C 180,E1 -11647.778,E2 -11647.778} C_VEL
LIN {X 0,Y 390.049,Z 703.897,A -85,B 0,C 180,E1 -11650.82,E2 -11650.82} C_VEL
LIN {X 0,Y 390.047,Z 703.896,A -85,B 0,C 180,E1 -11653.885,E2 -11653.885} C_VEL
LIN {X 0,Y 390.051,Z 703.894,A -85,B 0,C 180,E1 -11656.789,E2 -11656.789} C_VEL
LIN {X 0,Y 390.048,Z 703.889,A -85,B 0,C 180,E1 -11659.559,E2 -11659.559} C_VEL
LIN {X 0,Y 390.036,Z 703.9,A -85,B 0,C 180,E1 -11662.448,E2 -11662.448} C_VEL
LIN {X 0,Y 390.074,Z 703.891,A -85,B 0,C 180,E1 -11666.046,E2 -11666.046} C_VEL
LIN {X 0,Y 390.041,Z 703.899,A -85,B 0,C 180,E1 -11669.867,E2 -11669.867} C_VEL
LIN {X 0,Y 390.103,Z 703.893,A -85,B 0,C 180,E1 -11673.231,E2 -11673.231} C_VEL
LIN {X 0,Y 390.095,Z 703.89,A -85,B 0,C 180,E1 -11676.75,E2 -11676.75} C_VEL
LIN {X 0,Y 390.092,Z 703.894,A -85,B 0,C 180,E1 -11679.982,E2 -11679.982} C_VEL
LIN {X 0,Y 390.129,Z 703.881,A -85,B 0,C 180,E1 -11683.248,E2 -11683.248} C_VEL
LIN {X 0,Y 390.182,Z 703.874,A -85,B 0,C 180,E1 -11686.561,E2 -11686.561} C_VEL
LIN {X 0,Y 390.156,Z 703.886,A -85,B 0,C 180,E1 -11689.623,E2 -11689.623} C_VEL
LIN {X 0,Y 390.289,Z 703.867,A -85,B 0,C 180,E1 -11692.759,E2 -11692.759} C_VEL
LIN {X 0,Y 390.214,Z 703.871,A -85,B 0,C 180,E1 -11694.833,E2 -11694.833} C_VEL
LIN {X 0,Y 390.409,Z 703.853,A -85,B 0,C 180,E1 -11697.937,E2 -11697.937} C_VEL
LIN {X 0,Y 390.537,Z 703.833,A -85,B 0,C 180,E1 -11700,E2 -11700} C_VEL
LIN {X 0,Y 390.303,Z 703.863,A -85,B 0,C 180,E1 -11703.097,E2 -11703.097} C_VEL
LIN {X 0,Y 390.295,Z 703.864,A -85,B 0,C 180,E1 -11706.695,E2 -11706.695} C_VEL
LIN {X 0,Y 390.194,Z 703.878,A -85,B 0,C 180,E1 -11709.329,E2 -11709.329} C_VEL
LIN {X 0,Y 390.159,Z 703.881,A -85,B 0,C 180,E1 -11712.484,E2 -11712.484} C_VEL
LIN {X 0,Y 390.127,Z 703.882,A -85,B 0,C 180,E1 -11715.678,E2 -11715.678} C_VEL
LIN {X 0,Y 390.093,Z 703.892,A -85,B 0,C 180,E1 -11718.923,E2 -11718.923} C_VEL
LIN {X 0,Y 390.026,Z 703.896,A -85,B 0,C 180,E1 -11722.235,E2 -11722.235} C_VEL
LIN {X 0,Y 390.107,Z 703.894,A -85,B 0,C 180,E1 -11725.744,E2 -11725.744} C_VEL
LIN {X 0,Y 390.048,Z 703.889,A -85,B 0,C 180,E1 -11729.111,E2 -11729.111} C_VEL
LIN {X 0,Y 390.034,Z 703.891,A -85,B 0,C 180,E1 -11732.723,E2 -11732.723} C_VEL
LIN {X 0,Y 390.049,Z 703.894,A -85,B 0,C 180,E1 -11735.827,E2 -11735.827} C_VEL
LIN {X 0,Y 390.064,Z 703.893,A -85,B 0,C 180,E1 -11739.22,E2 -11739.22} C_VEL
LIN {X 0,Y 390.036,Z 703.901,A -85,B 0,C 180,E1 -11742.376,E2 -11742.376} C_VEL
LIN {X 0,Y 390.063,Z 704.122,A -85,B 0,C 180,E1 -11744.643,E2 -11744.643} C_VEL
LIN {X 0,Y 390.366,Z 705.349,A -85,B 0,C 180,E1 -11744.819,E2 -11744.819} C_VEL
LIN {X 0,Y 397.189,Z 721.453,A -85,B 0,C 180,E1 -11745.551,E2 -11745.551} C_VEL
LIN {X 0,Y 397.622,Z 722.538,A -85,B 0,C 180,E1 -11745.596,E2 -11745.596} C_VEL
LIN {X 0,Y 396.966,Z 783.579,A -85,B 0,C 180,E1 -11746.757,E2 -11746.757} C_VEL
LIN {X 0,Y 396.85,Z 796.932,A -85,B 0,C 180,E1 -11747.168,E2 -11747.168} C_VEL
LIN {X 0,Y 396.638,Z 809.15,A -85,B 0,C 180,E1 -11747.759,E2 -11747.759} C_VEL
LIN {X 0,Y 396.149,Z 821.36,A -85,B 0,C 180,E1 -11748.561,E2 -11748.561} C_VEL
LIN {X 0,Y 395.492,Z 832.123,A -85,B 0,C 180,E1 -11749.472,E2 -11749.472} C_VEL
LIN {X 0,Y 394.857,Z 841.712,A -85,B 0,C 180,E1 -11750.485,E2 -11750.485} C_VEL
LIN {X 0,Y 394.051,Z 851.082,A -85,B 0,C 180,E1 -11751.698,E2 -11751.698} C_VEL
LIN {X 0,Y 393.163,Z 860.202,A -85,B 0,C 180,E1 -11753.164,E2 -11753.164} C_VEL
LIN {X 0,Y 392.431,Z 867.973,A -85,B 0,C 180,E1 -11754.723,E2 -11754.723} C_VEL
LIN {X 0,Y 391.805,Z 873.937,A -85,B 0,C 180,E1 -11756.218,E2 -11756.218} C_VEL
LIN {X 0,Y 391.162,Z 879.67,A -85,B 0,C 180,E1 -11758.082,E2 -11758.082} C_VEL
LIN {X 0,Y 390.763,Z 883.492,A -85,B 0,C 180,E1 -11759.764,E2 -11759.764} C_VEL
LIN {X 0,Y 390.53,Z 885.472,A -85,B 0,C 180,E1 -11760.931,E2 -11760.931} C_VEL
LIN {X 0,Y 390.369,Z 886.87,A -85,B 0,C 180,E1 -11762.092,E2 -11762.092} C_VEL
LIN {X 0,Y 390.245,Z 887.801,A -85,B 0,C 180,E1 -11763.244,E2 -11763.244} C_VEL
LIN {X 0,Y 390.168,Z 888.21,A -85,B 0,C 180,E1 -11764.388,E2 -11764.388} C_VEL
LIN {X 0,Y 390.126,Z 888.158,A -85,B 0,C 180,E1 -11765.524,E2 -11765.524} C_VEL
LIN {X 0,Y 390.147,Z 887.598,A -85,B 0,C 180,E1 -11766.738,E2 -11766.738} C_VEL
LIN {X 0,Y 390.225,Z 886.657,A -85,B 0,C 180,E1 -11767.779,E2 -11767.779} C_VEL
LIN {X 0,Y 390.443,Z 884.417,A -85,B 0,C 180,E1 -11769.392,E2 -11769.392} C_VEL
LIN {X 0,Y 390.803,Z 880.877,A -85,B 0,C 180,E1 -11771.115,E2 -11771.115} C_VEL
LIN {X 0,Y 391.224,Z 876.227,A -85,B 0,C 180,E1 -11772.782,E2 -11772.782} C_VEL
LIN {X 0,Y 391.767,Z 870.438,A -85,B 0,C 180,E1 -11774.392,E2 -11774.392} C_VEL
LIN {X 0,Y 392.432,Z 863.046,A -85,B 0,C 180,E1 -11776.011,E2 -11776.011} C_VEL
LIN {X 0,Y 393.242,Z 853.823,A -85,B 0,C 180,E1 -11777.618,E2 -11777.618} C_VEL
LIN {X 0,Y 393.94,Z 844.841,A -85,B 0,C 180,E1 -11778.879,E2 -11778.879} C_VEL
LIN {X 0,Y 394.722,Z 833.668,A -85,B 0,C 180,E1 -11780.134,E2 -11780.134} C_VEL
LIN {X 0,Y 395.438,Z 821.831,A -85,B 0,C 180,E1 -11781.184,E2 -11781.184} C_VEL
LIN {X 0,Y 395.937,Z 809.283,A -85,B 0,C 180,E1 -11782.03,E2 -11782.03} C_VEL
LIN {X 0,Y 396.243,Z 796.18,A -85,B 0,C 180,E1 -11782.677,E2 -11782.677} C_VEL
LIN {X 0,Y 396.365,Z 783.094,A -85,B 0,C 180,E1 -11783.096,E2 -11783.096} C_VEL
LIN {X 0,Y 396.964,Z 721.535,A -85,B 0,C 180,E1 -11784.255,E2 -11784.255} C_VEL
LIN {X 0,Y 390.401,Z 704.868,A -85,B 0,C 180,E1 -11784.934,E2 -11784.934} C_VEL
LIN {X 0,Y 390.19,Z 703.99,A -85,B 0,C 180,E1 -11785.126,E2 -11785.126} C_VEL
LIN {X 0,Y 390.41,Z 703.854,A -85,B 0,C 180,E1 -11787.938,E2 -11787.938} C_VEL
LIN {X 0,Y 390.307,Z 703.866,A -85,B 0,C 180,E1 -11788.738,E2 -11788.738} C_VEL
LIN {X 0,Y 389.615,Z 703.956,A -85,B 0,C 180,E1 -11789.6,E2 -11789.6} C_VEL
LIN {X 0,Y 386.795,Z 704.312,A -85,B 0,C 180,E1 -11791.001,E2 -11791.001} C_VEL
LIN {X 0,Y 384.381,Z 704.611,A -85,B 0,C 180,E1 -11792.132,E2 -11792.132} C_VEL
LIN {X 0,Y 383.276,Z 704.744,A -85,B 0,C 180,E1 -11793.006,E2 -11793.006} C_VEL
LIN {X 0,Y 383.148,Z 704.758,A -85,B 0,C 180,E1 -11793.303,E2 -11793.303} C_VEL
LIN {X 0,Y 383.238,Z 704.749,A -85,B 0,C 180,E1 -11796.319,E2 -11796.319} C_VEL
LIN {X 0,Y 383.14,Z 704.757,A -85,B 0,C 180,E1 -11799.504,E2 -11799.504} C_VEL
LIN {X 0,Y 383.131,Z 704.756,A -85,B 0,C 180,E1 -11803.537,E2 -11803.537} C_VEL
LIN {X 0,Y 383.08,Z 704.765,A -85,B 0,C 180,E1 -11807.445,E2 -11807.445} C_VEL
LIN {X 0,Y 383.02,Z 704.763,A -85,B 0,C 180,E1 -11810.642,E2 -11810.642} C_VEL
LIN {X 0,Y 383.014,Z 704.772,A -85,B 0,C 180,E1 -11813.81,E2 -11813.81} C_VEL
LIN {X 0,Y 382.97,Z 704.768,A -85,B 0,C 180,E1 -11817.31,E2 -11817.31} C_VEL
LIN {X 0,Y 382.984,Z 704.78,A -85,B 0,C 180,E1 -11820.92,E2 -11820.92} C_VEL
LIN {X 0,Y 383.017,Z 704.752,A -85,B 0,C 180,E1 -11824.67,E2 -11824.67} C_VEL
LIN {X 0,Y 382.996,Z 704.774,A -85,B 0,C 180,E1 -11827.902,E2 -11827.902} C_VEL
LIN {X 0,Y 382.963,Z 704.783,A -85,B 0,C 180,E1 -11831.352,E2 -11831.352} C_VEL
LIN {X 0,Y 382.97,Z 704.778,A -85,B 0,C 180,E1 -11834.299,E2 -11834.299} C_VEL
LIN {X 0,Y 382.988,Z 704.778,A -85,B 0,C 180,E1 -11837.237,E2 -11837.237} C_VEL
LIN {X 0,Y 382.99,Z 704.778,A -85,B 0,C 180,E1 -11840.42,E2 -11840.42} C_VEL
LIN {X 0,Y 383.013,Z 704.776,A -85,B 0,C 180,E1 -11844.043,E2 -11844.043} C_VEL
LIN {X 0,Y 383.054,Z 704.92,A -85,B 0,C 180,E1 -11847.26,E2 -11847.26} C_VEL
LIN {X 0,Y 383.214,Z 705.711,A -85,B 0,C 180,E1 -11847.425,E2 -11847.425} C_VEL
LIN {X 0,Y 388.991,Z 721.973,A -85,B 0,C 180,E1 -11848.069,E2 -11848.069} C_VEL
LIN {X 0,Y 388.065,Z 781.613,A -85,B 0,C 180,E1 -11849.364,E2 -11849.364} C_VEL
LIN {X 0,Y 387.86,Z 792.916,A -85,B 0,C 180,E1 -11849.76,E2 -11849.76} C_VEL
LIN {X 0,Y 387.593,Z 803.84,A -85,B 0,C 180,E1 -11850.297,E2 -11850.297} C_VEL
LIN {X 0,Y 387.191,Z 814.122,A -85,B 0,C 180,E1 -11850.951,E2 -11850.951} C_VEL
LIN {X 0,Y 386.755,Z 823.145,A -85,B 0,C 180,E1 -11851.657,E2 -11851.657} C_VEL
LIN {X 0,Y 386.275,Z 832.1,A -85,B 0,C 180,E1 -11852.504,E2 -11852.504} C_VEL
LIN {X 0,Y 385.663,Z 841.504,A -85,B 0,C 180,E1 -11853.579,E2 -11853.579} C_VEL
LIN {X 0,Y 385.241,Z 849.095,A -85,B 0,C 180,E1 -11854.614,E2 -11854.614} C_VEL
LIN {X 0,Y 384.835,Z 855.71,A -85,B 0,C 180,E1 -11855.662,E2 -11855.662} C_VEL
LIN {X 0,Y 384.21,Z 863.366,A -85,B 0,C 180,E1 -11857.126,E2 -11857.126} C_VEL
LIN {X 0,Y 383.773,Z 869.345,A -85,B 0,C 180,E1 -11858.515,E2 -11858.515} C_VEL
LIN {X 0,Y 383.573,Z 873.413,A -85,B 0,C 180,E1 -11859.627,E2 -11859.627} C_VEL
LIN {X 0,Y 383.243,Z 878.206,A -85,B 0,C 180,E1 -11861.281,E2 -11861.281} C_VEL
LIN {X 0,Y 383.06,Z 881.785,A -85,B 0,C 180,E1 -11862.929,E2 -11862.929} C_VEL
LIN {X 0,Y 382.933,Z 883.622,A -85,B 0,C 180,E1 -11864.02,E2 -11864.02} C_VEL
LIN {X 0,Y 382.909,Z 885.784,A -85,B 0,C 180,E1 -11866.196,E2 -11866.196} C_VEL
LIN {X 0,Y 382.949,Z 886.233,A -85,B 0,C 180,E1 -11867.277,E2 -11867.277} C_VEL
LIN {X 0,Y 383.038,Z 886.202,A -85,B 0,C 180,E1 -11868.356,E2 -11868.356} C_VEL
LIN {X 0,Y 383.293,Z 884.888,A -85,B 0,C 180,E1 -11870.501,E2 -11870.501} C_VEL
LIN {X 0,Y 383.547,Z 883.309,A -85,B 0,C 180,E1 -11871.689,E2 -11871.689} C_VEL
LIN {X 0,Y 384.024,Z 879.562,A -85,B 0,C 180,E1 -11873.696,E2 -11873.696} C_VEL
LIN {X 0,Y 384.496,Z 875.268,A -85,B 0,C 180,E1 -11875.282,E2 -11875.282} C_VEL
LIN {X 0,Y 385.032,Z 869.713,A -85,B 0,C 180,E1 -11876.861,E2 -11876.861} C_VEL
LIN {X 0,Y 385.662,Z 864.038,A -85,B 0,C 180,E1 -11878.172,E2 -11878.172} C_VEL
LIN {X 0,Y 386.403,Z 857.162,A -85,B 0,C 180,E1 -11879.479,E2 -11879.479} C_VEL
LIN {X 0,Y 387.051,Z 850.136,A -85,B 0,C 180,E1 -11880.602,E2 -11880.602} C_VEL
LIN {X 0,Y 387.806,Z 840.863,A -85,B 0,C 180,E1 -11881.817,E2 -11881.817} C_VEL
LIN {X 0,Y 388.477,Z 832.525,A -85,B 0,C 180,E1 -11882.722,E2 -11882.722} C_VEL
LIN {X 0,Y 388.977,Z 824.077,A -85,B 0,C 180,E1 -11883.496,E2 -11883.496} C_VEL
LIN {X 0,Y 389.451,Z 813.611,A -85,B 0,C 180,E1 -11884.269,E2 -11884.269} C_VEL
LIN {X 0,Y 389.854,Z 802.95,A -85,B 0,C 180,E1 -11884.88,E2 -11884.88} C_VEL
LIN {X 0,Y 390.111,Z 792.598,A -85,B 0,C 180,E1 -11885.325,E2 -11885.325} C_VEL
LIN {X 0,Y 390.178,Z 779.588,A -85,B 0,C 180,E1 -11885.717,E2 -11885.717} C_VEL
LIN {X 0,Y 391.576,Z 723.849,A -85,B 0,C 180,E1 -11887.009,E2 -11887.009} C_VEL
LIN {X 0,Y 387.523,Z 714.225,A -85,B 0,C 180,E1 -11887.564,E2 -11887.564} C_VEL
LIN {X 0,Y 383.397,Z 705.727,A -85,B 0,C 180,E1 -11888.156,E2 -11888.156} C_VEL
LIN {X 0,Y 383.213,Z 704.822,A -85,B 0,C 180,E1 -11888.392,E2 -11888.392} C_VEL
LIN {X 0,Y 383.104,Z 704.762,A -85,B 0,C 180,E1 -11891.642,E2 -11891.642} C_VEL
LIN {X 0,Y 383.118,Z 704.763,A -85,B 0,C 180,E1 -11894.881,E2 -11894.881} C_VEL
LIN {X 0,Y 383.06,Z 704.771,A -85,B 0,C 180,E1 -11898.174,E2 -11898.174} C_VEL
LIN {X 0,Y 383,Z 704.776,A -85,B 0,C 180,E1 -11901.531,E2 -11901.531} C_VEL
LIN {X 0,Y 383.036,Z 704.772,A -85,B 0,C 180,E1 -11904.961,E2 -11904.961} C_VEL
LIN {X 0,Y 383.009,Z 704.776,A -85,B 0,C 180,E1 -11908.495,E2 -11908.495} C_VEL
LIN {X 0,Y 383.016,Z 704.774,A -85,B 0,C 180,E1 -11912.149,E2 -11912.149} C_VEL
LIN {X 0,Y 383.025,Z 704.772,A -85,B 0,C 180,E1 -11914.667,E2 -11914.667} C_VEL
LIN {X 0,Y 383.006,Z 704.775,A -85,B 0,C 180,E1 -11917.903,E2 -11917.903} C_VEL
LIN {X 0,Y 382.991,Z 704.778,A -85,B 0,C 180,E1 -11921.347,E2 -11921.347} C_VEL
LIN {X 0,Y 383.002,Z 704.776,A -85,B 0,C 180,E1 -11924.302,E2 -11924.302} C_VEL
LIN {X 0,Y 383.016,Z 704.774,A -85,B 0,C 180,E1 -11927.239,E2 -11927.239} C_VEL
LIN {X 0,Y 383.019,Z 704.772,A -85,B 0,C 180,E1 -11930.413,E2 -11930.413} C_VEL
LIN {X 0,Y 383.03,Z 704.773,A -85,B 0,C 180,E1 -11934.043,E2 -11934.043} C_VEL
LIN {X 0,Y 383.056,Z 704.979,A -85,B 0,C 180,E1 -11935.692,E2 -11935.692} C_VEL
LIN {X 0,Y 386.672,Z 720.127,A -85,B 0,C 180,E1 -11938.678,E2 -11938.678} C_VEL
LIN {X 0,Y 389.049,Z 731.583,A -85,B 0,C 180,E1 -11940.806,E2 -11940.806} C_VEL
LIN {X 0,Y 387.385,Z 750.279,A -85,B 0,C 180,E1 -11943.898,E2 -11943.898} C_VEL
LIN {X 0,Y 385.976,Z 768.921,A -85,B 0,C 180,E1 -11946.952,E2 -11946.952} C_VEL
LIN {X 0,Y 385.165,Z 780.518,A -85,B 0,C 180,E1 -11948.805,E2 -11948.805} C_VEL
LIN {X 0,Y 386.936,Z 795.441,A -85,B 0,C 180,E1 -11949.342,E2 -11949.342} C_VEL
LIN {X 0,Y 389.494,Z 826.643,A -85,B 0,C 180,E1 -11950.303,E2 -11950.303} C_VEL
LIN {X 0,Y 388.496,Z 893.537,A -85,B 0,C 180,E1 -11951.576,E2 -11951.576} C_VEL
LIN {X 0,Y 387.929,Z 906.805,A -85,B 0,C 180,E1 -11952.027,E2 -11952.027} C_VEL
LIN {X 0,Y 386.989,Z 920.123,A -85,B 0,C 180,E1 -11952.698,E2 -11952.698} C_VEL
LIN {X 0,Y 386.088,Z 931.354,A -85,B 0,C 180,E1 -11953.474,E2 -11953.474} C_VEL
LIN {X 0,Y 385.062,Z 943.055,A -85,B 0,C 180,E1 -11954.517,E2 -11954.517} C_VEL
LIN {X 0,Y 384.216,Z 953.731,A -85,B 0,C 180,E1 -11955.713,E2 -11955.713} C_VEL
LIN {X 0,Y 383.528,Z 963.201,A -85,B 0,C 180,E1 -11957.026,E2 -11957.026} C_VEL
LIN {X 0,Y 382.863,Z 971.041,A -85,B 0,C 180,E1 -11958.349,E2 -11958.349} C_VEL
LIN {X 0,Y 382.422,Z 978.751,A -85,B 0,C 180,E1 -11959.944,E2 -11959.944} C_VEL
LIN {X 0,Y 382.238,Z 984.976,A -85,B 0,C 180,E1 -11961.54,E2 -11961.54} C_VEL
LIN {X 0,Y 382.165,Z 990.221,A -85,B 0,C 180,E1 -11963.246,E2 -11963.246} C_VEL
LIN {X 0,Y 382.238,Z 993.695,A -85,B 0,C 180,E1 -11964.724,E2 -11964.724} C_VEL
LIN {X 0,Y 382.389,Z 995.659,A -85,B 0,C 180,E1 -11965.782,E2 -11965.782} C_VEL
LIN {X 0,Y 382.377,Z 997.13,A -85,B 0,C 180,E1 -11966.838,E2 -11966.838} C_VEL
LIN {X 0,Y 382.402,Z 998.161,A -85,B 0,C 180,E1 -11967.892,E2 -11967.892} C_VEL
LIN {X 0,Y 382.446,Z 998.788,A -85,B 0,C 180,E1 -11968.945,E2 -11968.945} C_VEL
LIN {X 0,Y 382.485,Z 999.009,A -85,B 0,C 180,E1 -11969.998,E2 -11969.998} C_VEL
LIN {X 0,Y 382.446,Z 998.78,A -85,B 0,C 180,E1 -11971.051,E2 -11971.051} C_VEL
LIN {X 0,Y 382.404,Z 998.123,A -85,B 0,C 180,E1 -11972.105,E2 -11972.105} C_VEL
LIN {X 0,Y 382.375,Z 997.061,A -85,B 0,C 180,E1 -11973.159,E2 -11973.159} C_VEL
LIN {X 0,Y 382.379,Z 995.592,A -85,B 0,C 180,E1 -11974.215,E2 -11974.215} C_VEL
LIN {X 0,Y 382.194,Z 992.482,A -85,B 0,C 180,E1 -11975.803,E2 -11975.803} C_VEL
LIN {X 0,Y 382.159,Z 988.321,A -85,B 0,C 180,E1 -11977.395,E2 -11977.395} C_VEL
LIN {X 0,Y 382.269,Z 981.982,A -85,B 0,C 180,E1 -11979.256,E2 -11979.256} C_VEL
LIN {X 0,Y 382.607,Z 975.092,A -85,B 0,C 180,E1 -11980.851,E2 -11980.851} C_VEL
LIN {X 0,Y 383.115,Z 966.585,A -85,B 0,C 180,E1 -11982.446,E2 -11982.446} C_VEL
LIN {X 0,Y 383.785,Z 959.795,A -85,B 0,C 180,E1 -11983.5,E2 -11983.5} C_VEL
LIN {X 0,Y 384.591,Z 949.664,A -85,B 0,C 180,E1 -11984.821,E2 -11984.821} C_VEL
LIN {X 0,Y 385.43,Z 939.763,A -85,B 0,C 180,E1 -11985.872,E2 -11985.872} C_VEL
LIN {X 0,Y 386.413,Z 929.122,A -85,B 0,C 180,E1 -11986.78,E2 -11986.78} C_VEL
LIN {X 0,Y 387.46,Z 916.374,A -85,B 0,C 180,E1 -11987.617,E2 -11987.617} C_VEL
LIN {X 0,Y 388.346,Z 902.948,A -85,B 0,C 180,E1 -11988.257,E2 -11988.257} C_VEL
LIN {X 0,Y 388.883,Z 890.578,A -85,B 0,C 180,E1 -11988.64,E2 -11988.64} C_VEL
LIN {X 0,Y 389.755,Z 823.785,A -85,B 0,C 180,E1 -11989.913,E2 -11989.913} C_VEL
LIN {X 0,Y 385.969,Z 788.107,A -85,B 0,C 180,E1 -11990.834,E2 -11990.834} C_VEL
LIN {X 0,Y 385.045,Z 780.806,A -85,B 0,C 180,E1 -11991.058,E2 -11991.058} C_VEL
LIN {X 0,Y 386.563,Z 760.525,A -85,B 0,C 180,E1 -11994.343,E2 -11994.343} C_VEL
LIN {X 0,Y 388.562,Z 736.489,A -85,B 0,C 180,E1 -11998.344,E2 -11998.344} C_VEL
LIN {X 0,Y 389.009,Z 731.456,A -85,B 0,C 180,E1 -11999.194,E2 -11999.194} C_VEL
LIN {X 0,Y 386.534,Z 719.481,A -85,B 0,C 180,E1 -12001.48,E2 -12001.48} C_VEL
LIN {X 0,Y 383.078,Z 704.956,A -85,B 0,C 180,E1 -12004.454,E2 -12004.454} C_VEL
LIN {X 0,Y 382.993,Z 704.776,A -85,B 0,C 180,E1 -12007.902,E2 -12007.902} C_VEL
LIN {X 0,Y 382.976,Z 704.78,A -85,B 0,C 180,E1 -12011.346,E2 -12011.346} C_VEL
LIN {X 0,Y 382.989,Z 704.778,A -85,B 0,C 180,E1 -12014.302,E2 -12014.302} C_VEL
LIN {X 0,Y 383.001,Z 704.777,A -85,B 0,C 180,E1 -12017.239,E2 -12017.239} C_VEL
LIN {X 0,Y 383.007,Z 704.765,A -85,B 0,C 180,E1 -12020.412,E2 -12020.412} C_VEL
LIN {X 0,Y 383.017,Z 704.764,A -85,B 0,C 180,E1 -12024.044,E2 -12024.044} C_VEL
LIN {X 0,Y 382.978,Z 704.779,A -85,B 0,C 180,E1 -12027.577,E2 -12027.577} C_VEL
LIN {X 0,Y 382.987,Z 704.777,A -85,B 0,C 180,E1 -12030.3,E2 -12030.3} C_VEL
LIN {X 0,Y 383.046,Z 704.767,A -85,B 0,C 180,E1 -12032.697,E2 -12032.697} C_VEL
LIN {X 0,Y 383.022,Z 704.772,A -85,B 0,C 180,E1 -12036.192,E2 -12036.192} C_VEL
LIN {X 0,Y 383.043,Z 704.769,A -85,B 0,C 180,E1 -12039.598,E2 -12039.598} C_VEL
LIN {X 0,Y 383.095,Z 704.756,A -85,B 0,C 180,E1 -12042.931,E2 -12042.931} C_VEL
LIN {X 0,Y 383.113,Z 704.754,A -85,B 0,C 180,E1 -12046.464,E2 -12046.464} C_VEL
LIN {X 0,Y 383.139,Z 704.751,A -85,B 0,C 180,E1 -12050.498,E2 -12050.498} C_VEL
LIN {X 0,Y 383.268,Z 704.743,A -85,B 0,C 180,E1 -12053.684,E2 -12053.684} C_VEL
LIN {X 0,Y 383.376,Z 704.729,A -85,B 0,C 180,E1 -12057.899,E2 -12057.899} C_VEL
LIN {X 0,Y 383.507,Z 704.708,A -85,B 0,C 180,E1 -12060,E2 -12060} C_VEL
LIN {X 0,Y 383.239,Z 704.743,A -85,B 0,C 180,E1 -12063.154,E2 -12063.154} C_VEL
LIN {X 0,Y 383.253,Z 704.742,A -85,B 0,C 180,E1 -12066.69,E2 -12066.69} C_VEL
LIN {X 0,Y 383.248,Z 704.742,A -85,B 0,C 180,E1 -12068.436,E2 -12068.436} C_VEL
LIN {X 0,Y 383.086,Z 704.761,A -85,B 0,C 180,E1 -12071.643,E2 -12071.643} C_VEL
LIN {X 0,Y 383.098,Z 704.765,A -85,B 0,C 180,E1 -12074.882,E2 -12074.882} C_VEL
LIN {X 0,Y 383.051,Z 704.768,A -85,B 0,C 180,E1 -12078.174,E2 -12078.174} C_VEL
LIN {X 0,Y 382.981,Z 704.776,A -85,B 0,C 180,E1 -12081.532,E2 -12081.532} C_VEL
LIN {X 0,Y 383.038,Z 704.765,A -85,B 0,C 180,E1 -12084.962,E2 -12084.962} C_VEL
LIN {X 0,Y 383.019,Z 704.763,A -85,B 0,C 180,E1 -12088.271,E2 -12088.271} C_VEL
LIN {X 0,Y 383,Z 704.769,A -85,B 0,C 180,E1 -12092.151,E2 -12092.151} C_VEL
LIN {X 0,Y 383.01,Z 704.775,A -85,B 0,C 180,E1 -12094.669,E2 -12094.669} C_VEL
LIN {X 0,Y 382.994,Z 704.777,A -85,B 0,C 180,E1 -12097.906,E2 -12097.906} C_VEL
LIN {X 0,Y 382.977,Z 704.777,A -85,B 0,C 180,E1 -12101.349,E2 -12101.349} C_VEL
LIN {X 0,Y 383.019,Z 704.958,A -85,B 0,C 180,E1 -12104.208,E2 -12104.208} C_VEL
LIN {X 0,Y 383.196,Z 705.799,A -85,B 0,C 180,E1 -12104.373,E2 -12104.373} C_VEL
LIN {X 0,Y 390.979,Z 724.174,A -85,B 0,C 180,E1 -12105.245,E2 -12105.245} C_VEL
LIN {X 0,Y 390.316,Z 784.485,A -85,B 0,C 180,E1 -12106.414,E2 -12106.414} C_VEL
LIN {X 0,Y 390.205,Z 798.207,A -85,B 0,C 180,E1 -12106.846,E2 -12106.846} C_VEL
LIN {X 0,Y 389.967,Z 810.364,A -85,B 0,C 180,E1 -12107.447,E2 -12107.447} C_VEL
LIN {X 0,Y 389.492,Z 821.764,A -85,B 0,C 180,E1 -12108.205,E2 -12108.205} C_VEL
LIN {X 0,Y 388.739,Z 833.668,A -85,B 0,C 180,E1 -12109.227,E2 -12109.227} C_VEL
LIN {X 0,Y 388.028,Z 843.713,A -85,B 0,C 180,E1 -12110.326,E2 -12110.326} C_VEL
LIN {X 0,Y 387.093,Z 853.609,A -85,B 0,C 180,E1 -12111.668,E2 -12111.668} C_VEL
LIN {X 0,Y 386.184,Z 862.689,A -85,B 0,C 180,E1 -12113.201,E2 -12113.201} C_VEL
LIN {X 0,Y 385.42,Z 870.211,A -85,B 0,C 180,E1 -12114.81,E2 -12114.81} C_VEL
LIN {X 0,Y 384.719,Z 876.335,A -85,B 0,C 180,E1 -12116.456,E2 -12116.456} C_VEL
LIN {X 0,Y 384.192,Z 880.751,A -85,B 0,C 180,E1 -12117.963,E2 -12117.963} C_VEL
LIN {X 0,Y 383.843,Z 883.985,A -85,B 0,C 180,E1 -12119.379,E2 -12119.379} C_VEL
LIN {X 0,Y 383.639,Z 885.733,A -85,B 0,C 180,E1 -12120.357,E2 -12120.357} C_VEL
LIN {X 0,Y 383.436,Z 887.48,A -85,B 0,C 180,E1 -12121.618,E2 -12121.618} C_VEL
LIN {X 0,Y 383.287,Z 888.486,A -85,B 0,C 180,E1 -12122.718,E2 -12122.718} C_VEL
LIN {X 0,Y 383.192,Z 889.145,A -85,B 0,C 180,E1 -12123.988,E2 -12123.988} C_VEL
LIN {X 0,Y 383.124,Z 889.262,A -85,B 0,C 180,E1 -12125.047,E2 -12125.047} C_VEL
LIN {X 0,Y 383.108,Z 888.751,A -85,B 0,C 180,E1 -12126.526,E2 -12126.526} C_VEL
LIN {X 0,Y 383.313,Z 886.866,A -85,B 0,C 180,E1 -12128.49,E2 -12128.49} C_VEL
LIN {X 0,Y 383.581,Z 884.093,A -85,B 0,C 180,E1 -12130.188,E2 -12130.188} C_VEL
LIN {X 0,Y 384.032,Z 879.574,A -85,B 0,C 180,E1 -12132.108,E2 -12132.108} C_VEL
LIN {X 0,Y 384.458,Z 875.127,A -85,B 0,C 180,E1 -12133.542,E2 -12133.542} C_VEL
LIN {X 0,Y 385.119,Z 868.333,A -85,B 0,C 180,E1 -12135.285,E2 -12135.285} C_VEL
LIN {X 0,Y 385.872,Z 860.616,A -85,B 0,C 180,E1 -12136.842,E2 -12136.842} C_VEL
LIN {X 0,Y 386.562,Z 852.368,A -85,B 0,C 180,E1 -12138.199,E2 -12138.199} C_VEL
LIN {X 0,Y 387.368,Z 842.284,A -85,B 0,C 180,E1 -12139.549,E2 -12139.549} C_VEL
LIN {X 0,Y 388.031,Z 832.369,A -85,B 0,C 180,E1 -12140.62,E2 -12140.62} C_VEL
LIN {X 0,Y 388.707,Z 821.517,A -85,B 0,C 180,E1 -12141.554,E2 -12141.554} C_VEL
LIN {X 0,Y 389.23,Z 808.603,A -85,B 0,C 180,E1 -12142.414,E2 -12142.414} C_VEL
LIN {X 0,Y 389.526,Z 795.646,A -85,B 0,C 180,E1 -12143.035,E2 -12143.035} C_VEL
LIN {X 0,Y 389.631,Z 782.036,A -85,B 0,C 180,E1 -12143.447,E2 -12143.447} C_VEL
LIN {X 0,Y 390.234,Z 723.05,A -85,B 0,C 180,E1 -12144.569,E2 -12144.569} C_VEL
LIN {X 0,Y 383.819,Z 707.08,A -85,B 0,C 180,E1 -12145.222,E2 -12145.222} C_VEL
LIN {X 0,Y 383.183,Z 705.295,A -85,B 0,C 180,E1 -12145.366,E2 -12145.366} C_VEL
LIN {X 0,Y 383.07,Z 704.775,A -85,B 0,C 180,E1 -12145.661,E2 -12145.661} C_VEL
LIN {X 0,Y 383.375,Z 704.73,A -85,B 0,C 180,E1 -12147.9,E2 -12147.9} C_VEL
LIN {X 0,Y 383.371,Z 704.729,A -85,B 0,C 180,E1 -12152.103,E2 -12152.103} C_VEL
LIN {X 0,Y 383.148,Z 704.758,A -85,B 0,C 180,E1 -12153.303,E2 -12153.303} C_VEL
LIN {X 0,Y 382.38,Z 704.854,A -85,B 0,C 180,E1 -12154.181,E2 -12154.181} C_VEL
LIN {X 0,Y 379.518,Z 705.211,A -85,B 0,C 180,E1 -12155.609,E2 -12155.609} C_VEL
LIN {X 0,Y 377.19,Z 705.497,A -85,B 0,C 180,E1 -12156.764,E2 -12156.764} C_VEL
LIN {X 0,Y 376.239,Z 705.613,A -85,B 0,C 180,E1 -12157.657,E2 -12157.657} C_VEL
LIN {X 0,Y 376.184,Z 705.621,A -85,B 0,C 180,E1 -12157.958,E2 -12157.958} C_VEL
LIN {X 0,Y 376.077,Z 705.634,A -85,B 0,C 180,E1 -12160.772,E2 -12160.772} C_VEL
LIN {X 0,Y 376.07,Z 705.637,A -85,B 0,C 180,E1 -12164.062,E2 -12164.062} C_VEL
LIN {X 0,Y 376.031,Z 705.642,A -85,B 0,C 180,E1 -12167.599,E2 -12167.599} C_VEL
LIN {X 0,Y 375.985,Z 705.64,A -85,B 0,C 180,E1 -12170.833,E2 -12170.833} C_VEL
LIN {X 0,Y 375.964,Z 705.65,A -85,B 0,C 180,E1 -12174.285,E2 -12174.285} C_VEL
LIN {X 0,Y 375.922,Z 705.649,A -85,B 0,C 180,E1 -12177.866,E2 -12177.866} C_VEL
LIN {X 0,Y 375.942,Z 705.655,A -85,B 0,C 180,E1 -12180.689,E2 -12180.689} C_VEL
LIN {X 0,Y 375.963,Z 705.631,A -85,B 0,C 180,E1 -12184.113,E2 -12184.113} C_VEL
LIN {X 0,Y 375.953,Z 705.639,A -85,B 0,C 180,E1 -12186.743,E2 -12186.743} C_VEL
LIN {X 0,Y 375.944,Z 705.654,A -85,B 0,C 180,E1 -12189.962,E2 -12189.962} C_VEL
LIN {X 0,Y 375.909,Z 705.663,A -85,B 0,C 180,E1 -12193.771,E2 -12193.771} C_VEL
LIN {X 0,Y 375.938,Z 705.654,A -85,B 0,C 180,E1 -12196.812,E2 -12196.812} C_VEL
LIN {X 0,Y 375.939,Z 705.656,A -85,B 0,C 180,E1 -12200.534,E2 -12200.534} C_VEL
LIN {X 0,Y 375.96,Z 705.655,A -85,B 0,C 180,E1 -12203.498,E2 -12203.498} C_VEL
LIN {X 0,Y 376.028,Z 705.863,A -85,B 0,C 180,E1 -12206.992,E2 -12206.992} C_VEL
LIN {X 0,Y 376.238,Z 706.813,A -85,B 0,C 180,E1 -12207.151,E2 -12207.151} C_VEL
LIN {X 0,Y 382.205,Z 723.797,A -85,B 0,C 180,E1 -12207.821,E2 -12207.821} C_VEL
LIN {X 0,Y 381.182,Z 782.021,A -85,B 0,C 180,E1 -12209.111,E2 -12209.111} C_VEL
LIN {X 0,Y 380.992,Z 793.886,A -85,B 0,C 180,E1 -12209.536,E2 -12209.536} C_VEL
LIN {X 0,Y 380.725,Z 803.891,A -85,B 0,C 180,E1 -12210.029,E2 -12210.029} C_VEL
LIN {X 0,Y 380.339,Z 814.163,A -85,B 0,C 180,E1 -12210.681,E2 -12210.681} C_VEL
LIN {X 0,Y 379.789,Z 824.911,A -85,B 0,C 180,E1 -12211.542,E2 -12211.542} C_VEL
LIN {X 0,Y 379.317,Z 833.743,A -85,B 0,C 180,E1 -12212.406,E2 -12212.406} C_VEL
LIN {X 0,Y 378.742,Z 841.993,A -85,B 0,C 180,E1 -12213.36,E2 -12213.36} C_VEL
LIN {X 0,Y 378.291,Z 849.648,A -85,B 0,C 180,E1 -12214.409,E2 -12214.409} C_VEL
LIN {X 0,Y 377.756,Z 857.728,A -85,B 0,C 180,E1 -12215.734,E2 -12215.734} C_VEL
LIN {X 0,Y 377.226,Z 864.086,A -85,B 0,C 180,E1 -12216.968,E2 -12216.968} C_VEL
LIN {X 0,Y 376.899,Z 869.091,A -85,B 0,C 180,E1 -12218.103,E2 -12218.103} C_VEL
LIN {X 0,Y 376.501,Z 875.096,A -85,B 0,C 180,E1 -12219.798,E2 -12219.798} C_VEL
LIN {X 0,Y 376.177,Z 879.748,A -85,B 0,C 180,E1 -12221.482,E2 -12221.482} C_VEL
LIN {X 0,Y 376.087,Z 882.27,A -85,B 0,C 180,E1 -12222.602,E2 -12222.602} C_VEL
LIN {X 0,Y 375.921,Z 884.131,A -85,B 0,C 180,E1 -12223.714,E2 -12223.714} C_VEL
LIN {X 0,Y 375.879,Z 886.661,A -85,B 0,C 180,E1 -12225.932,E2 -12225.932} C_VEL
LIN {X 0,Y 375.915,Z 887.208,A -85,B 0,C 180,E1 -12227.035,E2 -12227.035} C_VEL
LIN {X 0,Y 376.001,Z 887.347,A -85,B 0,C 180,E1 -12228.135,E2 -12228.135} C_VEL
LIN {X 0,Y 376.14,Z 887.008,A -85,B 0,C 180,E1 -12229.231,E2 -12229.231} C_VEL
LIN {X 0,Y 376.271,Z 886.219,A -85,B 0,C 180,E1 -12230.322,E2 -12230.322} C_VEL
LIN {X 0,Y 376.715,Z 883.416,A -85,B 0,C 180,E1 -12232.496,E2 -12232.496} C_VEL
LIN {X 0,Y 377.187,Z 880.079,A -85,B 0,C 180,E1 -12234.118,E2 -12234.118} C_VEL
LIN {X 0,Y 377.691,Z 875.628,A -85,B 0,C 180,E1 -12235.731,E2 -12235.731} C_VEL
LIN {X 0,Y 378.191,Z 871.012,A -85,B 0,C 180,E1 -12237.071,E2 -12237.071} C_VEL
LIN {X 0,Y 378.864,Z 865.367,A -85,B 0,C 180,E1 -12238.405,E2 -12238.405} C_VEL
LIN {X 0,Y 379.645,Z 858.669,A -85,B 0,C 180,E1 -12239.708,E2 -12239.708} C_VEL
LIN {X 0,Y 380.447,Z 850.217,A -85,B 0,C 180,E1 -12241.058,E2 -12241.058} C_VEL
LIN {X 0,Y 381.133,Z 842.269,A -85,B 0,C 180,E1 -12242.113,E2 -12242.113} C_VEL
LIN {X 0,Y 381.824,Z 833.98,A -85,B 0,C 180,E1 -12243.033,E2 -12243.033} C_VEL
LIN {X 0,Y 382.482,Z 823.973,A -85,B 0,C 180,E1 -12243.951,E2 -12243.951} C_VEL
LIN {X 0,Y 382.942,Z 814.3,A -85,B 0,C 180,E1 -12244.671,E2 -12244.671} C_VEL
LIN {X 0,Y 383.355,Z 804.247,A -85,B 0,C 180,E1 -12245.259,E2 -12245.259} C_VEL
LIN {X 0,Y 383.628,Z 793.911,A -85,B 0,C 180,E1 -12245.717,E2 -12245.717} C_VEL
LIN {X 0,Y 383.706,Z 781.228,A -85,B 0,C 180,E1 -12246.111,E2 -12246.111} C_VEL
LIN {X 0,Y 385.125,Z 725.538,A -85,B 0,C 180,E1 -12247.444,E2 -12247.444} C_VEL
LIN {X 0,Y 381.566,Z 717.16,A -85,B 0,C 180,E1 -12247.957,E2 -12247.957} C_VEL
LIN {X 0,Y 376.278,Z 706.474,A -85,B 0,C 180,E1 -12248.736,E2 -12248.736} C_VEL
LIN {X 0,Y 376.136,Z 705.706,A -85,B 0,C 180,E1 -12248.962,E2 -12248.962} C_VEL
LIN {X 0,Y 376.111,Z 705.635,A -85,B 0,C 180,E1 -12252.958,E2 -12252.958} C_VEL
LIN {X 0,Y 376.033,Z 705.646,A -85,B 0,C 180,E1 -12256.281,E2 -12256.281} C_VEL
LIN {X 0,Y 376.004,Z 705.649,A -85,B 0,C 180,E1 -12259.66,E2 -12259.66} C_VEL
LIN {X 0,Y 375.985,Z 705.649,A -85,B 0,C 180,E1 -12263.661,E2 -12263.661} C_VEL
LIN {X 0,Y 375.971,Z 705.653,A -85,B 0,C 180,E1 -12266.656,E2 -12266.656} C_VEL
LIN {X 0,Y 375.97,Z 705.653,A -85,B 0,C 180,E1 -12270.312,E2 -12270.312} C_VEL
LIN {X 0,Y 375.967,Z 705.652,A -85,B 0,C 180,E1 -12274.111,E2 -12274.111} C_VEL
LIN {X 0,Y 375.96,Z 705.652,A -85,B 0,C 180,E1 -12276.74,E2 -12276.74} C_VEL
LIN {X 0,Y 375.995,Z 705.649,A -85,B 0,C 180,E1 -12279.97,E2 -12279.97} C_VEL
LIN {X 0,Y 375.936,Z 705.658,A -85,B 0,C 180,E1 -12283.765,E2 -12283.765} C_VEL
LIN {X 0,Y 375.94,Z 705.656,A -85,B 0,C 180,E1 -12286.81,E2 -12286.81} C_VEL
LIN {X 0,Y 375.966,Z 705.651,A -85,B 0,C 180,E1 -12290.536,E2 -12290.536} C_VEL
LIN {X 0,Y 375.969,Z 705.655,A -85,B 0,C 180,E1 -12293.495,E2 -12293.495} C_VEL
LIN {X 0,Y 376.028,Z 705.891,A -85,B 0,C 180,E1 -12295.349,E2 -12295.349} C_VEL
LIN {X 0,Y 379.879,Z 722.13,A -85,B 0,C 180,E1 -12298.605,E2 -12298.605} C_VEL
LIN {X 0,Y 382.023,Z 732.231,A -85,B 0,C 180,E1 -12300.519,E2 -12300.519} C_VEL
LIN {X 0,Y 381.306,Z 742.194,A -85,B 0,C 180,E1 -12302.216,E2 -12302.216} C_VEL
LIN {X 0,Y 379.26,Z 766.163,A -85,B 0,C 180,E1 -12306.23,E2 -12306.23} C_VEL
LIN {X 0,Y 378.346,Z 778.484,A -85,B 0,C 180,E1 -12308.246,E2 -12308.246} C_VEL
LIN {X 0,Y 380.417,Z 795.384,A -85,B 0,C 180,E1 -12308.889,E2 -12308.889} C_VEL
LIN {X 0,Y 382.967,Z 827.297,A -85,B 0,C 180,E1 -12309.901,E2 -12309.901} C_VEL
LIN {X 0,Y 382.348,Z 854.302,A -85,B 0,C 180,E1 -12310.508,E2 -12310.508} C_VEL
LIN {X 0,Y 381.687,Z 893.011,A -85,B 0,C 180,E1 -12311.27,E2 -12311.27} C_VEL
LIN {X 0,Y 381.109,Z 906.125,A -85,B 0,C 180,E1 -12311.728,E2 -12311.728} C_VEL
LIN {X 0,Y 380.217,Z 918.804,A -85,B 0,C 180,E1 -12312.38,E2 -12312.38} C_VEL
LIN {X 0,Y 379.262,Z 930.124,A -85,B 0,C 180,E1 -12313.168,E2 -12313.168} C_VEL
LIN {X 0,Y 378.176,Z 941.864,A -85,B 0,C 180,E1 -12314.228,E2 -12314.228} C_VEL
LIN {X 0,Y 377.242,Z 952.91,A -85,B 0,C 180,E1 -12315.487,E2 -12315.487} C_VEL
LIN {X 0,Y 376.582,Z 962.079,A -85,B 0,C 180,E1 -12316.783,E2 -12316.783} C_VEL
LIN {X 0,Y 375.855,Z 969.936,A -85,B 0,C 180,E1 -12318.129,E2 -12318.129} C_VEL
LIN {X 0,Y 375.366,Z 977.665,A -85,B 0,C 180,E1 -12319.753,E2 -12319.753} C_VEL
LIN {X 0,Y 375.161,Z 983.908,A -85,B 0,C 180,E1 -12321.379,E2 -12321.379} C_VEL
LIN {X 0,Y 375.109,Z 989.446,A -85,B 0,C 180,E1 -12323.219,E2 -12323.219} C_VEL
LIN {X 0,Y 375.166,Z 992.657,A -85,B 0,C 180,E1 -12324.624,E2 -12324.624} C_VEL
LIN {X 0,Y 375.319,Z 994.627,A -85,B 0,C 180,E1 -12325.703,E2 -12325.703} C_VEL
LIN {X 0,Y 375.334,Z 996.11,A -85,B 0,C 180,E1 -12326.778,E2 -12326.778} C_VEL
LIN {X 0,Y 375.364,Z 997.145,A -85,B 0,C 180,E1 -12327.852,E2 -12327.852} C_VEL
LIN {X 0,Y 375.413,Z 997.775,A -85,B 0,C 180,E1 -12328.926,E2 -12328.926} C_VEL
LIN {X 0,Y 375.456,Z 997.999,A -85,B 0,C 180,E1 -12329.998,E2 -12329.998} C_VEL
LIN {X 0,Y 375.412,Z 997.775,A -85,B 0,C 180,E1 -12331.071,E2 -12331.071} C_VEL
LIN {X 0,Y 375.363,Z 997.117,A -85,B 0,C 180,E1 -12332.144,E2 -12332.144} C_VEL
LIN {X 0,Y 375.33,Z 996.057,A -85,B 0,C 180,E1 -12333.219,E2 -12333.219} C_VEL
LIN {X 0,Y 375.31,Z 994.585,A -85,B 0,C 180,E1 -12334.294,E2 -12334.294} C_VEL
LIN {X 0,Y 375.14,Z 991.483,A -85,B 0,C 180,E1 -12335.913,E2 -12335.913} C_VEL
LIN {X 0,Y 375.11,Z 987.328,A -85,B 0,C 180,E1 -12337.534,E2 -12337.534} C_VEL
LIN {X 0,Y 375.22,Z 980.997,A -85,B 0,C 180,E1 -12339.431,E2 -12339.431} C_VEL
LIN {X 0,Y 375.585,Z 974.115,A -85,B 0,C 180,E1 -12341.056,E2 -12341.056} C_VEL
LIN {X 0,Y 376.142,Z 965.618,A -85,B 0,C 180,E1 -12342.68,E2 -12342.68} C_VEL
LIN {X 0,Y 376.751,Z 958.83,A -85,B 0,C 180,E1 -12343.757,E2 -12343.757} C_VEL
LIN {X 0,Y 377.635,Z 948.72,A -85,B 0,C 180,E1 -12345.101,E2 -12345.101} C_VEL
LIN {X 0,Y 378.569,Z 938.849,A -85,B 0,C 180,E1 -12346.167,E2 -12346.167} C_VEL
LIN {X 0,Y 379.592,Z 928.253,A -85,B 0,C 180,E1 -12347.091,E2 -12347.091} C_VEL
LIN {X 0,Y 380.679,Z 915.563,A -85,B 0,C 180,E1 -12347.942,E2 -12347.942} C_VEL
LIN {X 0,Y 381.602,Z 902.237,A -85,B 0,C 180,E1 -12348.591,E2 -12348.591} C_VEL
LIN {X 0,Y 382.192,Z 888.742,A -85,B 0,C 180,E1 -12349.014,E2 -12349.014} C_VEL
LIN {X 0,Y 383.1,Z 824.613,A -85,B 0,C 180,E1 -12350.257,E2 -12350.257} C_VEL
LIN {X 0,Y 379.298,Z 788.651,A -85,B 0,C 180,E1 -12351.204,E2 -12351.204} C_VEL
LIN {X 0,Y 378.159,Z 779.81,A -85,B 0,C 180,E1 -12351.473,E2 -12351.473} C_VEL
LIN {X 0,Y 379.633,Z 761.3,A -85,B 0,C 180,E1 -12354.526,E2 -12354.526} C_VEL
LIN {X 0,Y 381.734,Z 737.33,A -85,B 0,C 180,E1 -12358.597,E2 -12358.597} C_VEL
LIN {X 0,Y 382.064,Z 732.293,A -85,B 0,C 180,E1 -12359.474,E2 -12359.474} C_VEL
LIN {X 0,Y 379.721,Z 721.246,A -85,B 0,C 180,E1 -12361.637,E2 -12361.637} C_VEL
LIN {X 0,Y 376.166,Z 706.495,A -85,B 0,C 180,E1 -12364.708,E2 -12364.708} C_VEL
LIN {X 0,Y 375.982,Z 705.69,A -85,B 0,C 180,E1 -12364.996,E2 -12364.996} C_VEL
LIN {X 0,Y 375.967,Z 705.651,A -85,B 0,C 180,E1 -12368.269,E2 -12368.269} C_VEL
LIN {X 0,Y 375.927,Z 705.658,A -85,B 0,C 180,E1 -12371.599,E2 -12371.599} C_VEL
LIN {X 0,Y 375.921,Z 705.655,A -85,B 0,C 180,E1 -12375.267,E2 -12375.267} C_VEL
LIN {X 0,Y 375.927,Z 705.659,A -85,B 0,C 180,E1 -12378.398,E2 -12378.398} C_VEL
LIN {X 0,Y 375.967,Z 705.652,A -85,B 0,C 180,E1 -12381.728,E2 -12381.728} C_VEL
LIN {X 0,Y 375.97,Z 705.642,A -85,B 0,C 180,E1 -12385.331,E2 -12385.331} C_VEL
LIN {X 0,Y 375.95,Z 705.652,A -85,B 0,C 180,E1 -12388.437,E2 -12388.437} C_VEL
LIN {X 0,Y 375.991,Z 705.646,A -85,B 0,C 180,E1 -12392.141,E2 -12392.141} C_VEL
LIN {X 0,Y 375.995,Z 705.645,A -85,B 0,C 180,E1 -12394.538,E2 -12394.538} C_VEL
LIN {X 0,Y 375.952,Z 705.649,A -85,B 0,C 180,E1 -12398.045,E2 -12398.045} C_VEL
LIN {X 0,Y 376.012,Z 705.648,A -85,B 0,C 180,E1 -12401.473,E2 -12401.473} C_VEL
LIN {X 0,Y 376.049,Z 705.64,A -85,B 0,C 180,E1 -12404.832,E2 -12404.832} C_VEL
LIN {X 0,Y 376.039,Z 705.646,A -85,B 0,C 180,E1 -12408.136,E2 -12408.136} C_VEL
LIN {X 0,Y 376.206,Z 705.616,A -85,B 0,C 180,E1 -12411.919,E2 -12411.919} C_VEL
LIN {X 0,Y 376.158,Z 705.624,A -85,B 0,C 180,E1 -12414.64,E2 -12414.64} C_VEL
LIN {X 0,Y 376.342,Z 705.604,A -85,B 0,C 180,E1 -12417.86,E2 -12417.86} C_VEL
LIN {X 0,Y 376.476,Z 705.584,A -85,B 0,C 180,E1 -12420,E2 -12420} C_VEL
LIN {X 0,Y 376.177,Z 705.622,A -85,B 0,C 180,E1 -12423.213,E2 -12423.213} C_VEL
LIN {X 0,Y 376.217,Z 705.62,A -85,B 0,C 180,E1 -12426.682,E2 -12426.682} C_VEL
LIN {X 0,Y 376.193,Z 705.62,A -85,B 0,C 180,E1 -12428.596,E2 -12428.596} C_VEL
LIN {X 0,Y 376.039,Z 705.639,A -85,B 0,C 180,E1 -12431.864,E2 -12431.864} C_VEL
LIN {X 0,Y 376.046,Z 705.639,A -85,B 0,C 180,E1 -12435.168,E2 -12435.168} C_VEL
LIN {X 0,Y 375.997,Z 705.649,A -85,B 0,C 180,E1 -12438.528,E2 -12438.528} C_VEL
LIN {X 0,Y 375.945,Z 705.65,A -85,B 0,C 180,E1 -12441.956,E2 -12441.956} C_VEL
LIN {X 0,Y 375.994,Z 705.649,A -85,B 0,C 180,E1 -12445.462,E2 -12445.462} C_VEL
LIN {X 0,Y 375.951,Z 705.644,A -85,B 0,C 180,E1 -12449.081,E2 -12449.081} C_VEL
LIN {X 0,Y 375.942,Z 705.647,A -85,B 0,C 180,E1 -12452.83,E2 -12452.83} C_VEL
LIN {X 0,Y 375.95,Z 705.651,A -85,B 0,C 180,E1 -12455.417,E2 -12455.417} C_VEL
LIN {X 0,Y 375.968,Z 705.648,A -85,B 0,C 180,E1 -12458.272,E2 -12458.272} C_VEL
LIN {X 0,Y 375.927,Z 705.656,A -85,B 0,C 180,E1 -12461.602,E2 -12461.602} C_VEL
LIN {X 0,Y 376.004,Z 705.797,A -85,B 0,C 180,E1 -12463.756,E2 -12463.756} C_VEL
LIN {X 0,Y 376.186,Z 706.725,A -85,B 0,C 180,E1 -12463.945,E2 -12463.945} C_VEL
LIN {X 0,Y 384.035,Z 725.01,A -85,B 0,C 180,E1 -12464.846,E2 -12464.846} C_VEL
LIN {X 0,Y 384.442,Z 726.468,A -85,B 0,C 180,E1 -12464.901,E2 -12464.901} C_VEL
LIN {X 0,Y 383.684,Z 783.109,A -85,B 0,C 180,E1 -12466.006,E2 -12466.006} C_VEL
LIN {X 0,Y 383.626,Z 796.7,A -85,B 0,C 180,E1 -12466.407,E2 -12466.407} C_VEL
LIN {X 0,Y 383.372,Z 809.423,A -85,B 0,C 180,E1 -12467,E2 -12467} C_VEL
LIN {X 0,Y 382.907,Z 821.22,A -85,B 0,C 180,E1 -12467.763,E2 -12467.763} C_VEL
LIN {X 0,Y 382.192,Z 832.356,A -85,B 0,C 180,E1 -12468.699,E2 -12468.699} C_VEL
LIN {X 0,Y 381.407,Z 843.088,A -85,B 0,C 180,E1 -12469.842,E2 -12469.842} C_VEL
LIN {X 0,Y 380.519,Z 852.648,A -85,B 0,C 180,E1 -12471.102,E2 -12471.102} C_VEL
LIN {X 0,Y 379.717,Z 860.419,A -85,B 0,C 180,E1 -12472.356,E2 -12472.356} C_VEL
LIN {X 0,Y 378.846,Z 868.285,A -85,B 0,C 180,E1 -12473.917,E2 -12473.917} C_VEL
LIN {X 0,Y 378.013,Z 875.708,A -85,B 0,C 180,E1 -12475.78,E2 -12475.78} C_VEL
LIN {X 0,Y 377.407,Z 880.481,A -85,B 0,C 180,E1 -12477.316,E2 -12477.316} C_VEL
LIN {X 0,Y 376.935,Z 884.629,A -85,B 0,C 180,E1 -12479.058,E2 -12479.058} C_VEL
LIN {X 0,Y 376.517,Z 887.791,A -85,B 0,C 180,E1 -12480.969,E2 -12480.969} C_VEL
LIN {X 0,Y 376.344,Z 889.116,A -85,B 0,C 180,E1 -12482.171,E2 -12482.171} C_VEL
LIN {X 0,Y 376.193,Z 890.075,A -85,B 0,C 180,E1 -12483.733,E2 -12483.733} C_VEL
LIN {X 0,Y 376.079,Z 890.135,A -85,B 0,C 180,E1 -12485.726,E2 -12485.726} C_VEL
LIN {X 0,Y 376.096,Z 889.516,A -85,B 0,C 180,E1 -12486.897,E2 -12486.897} C_VEL
LIN {X 0,Y 376.355,Z 887.207,A -85,B 0,C 180,E1 -12489.019,E2 -12489.019} C_VEL
LIN {X 0,Y 376.728,Z 883.709,A -85,B 0,C 180,E1 -12490.947,E2 -12490.947} C_VEL
LIN {X 0,Y 377.169,Z 879.355,A -85,B 0,C 180,E1 -12492.656,E2 -12492.656} C_VEL
LIN {X 0,Y 377.752,Z 873.737,A -85,B 0,C 180,E1 -12494.351,E2 -12494.351} C_VEL
LIN {X 0,Y 378.422,Z 866.714,A -85,B 0,C 180,E1 -12496.031,E2 -12496.031} C_VEL
LIN {X 0,Y 379.181,Z 859.487,A -85,B 0,C 180,E1 -12497.423,E2 -12497.423} C_VEL
LIN {X 0,Y 379.988,Z 850.131,A -85,B 0,C 180,E1 -12498.893,E2 -12498.893} C_VEL
LIN {X 0,Y 380.785,Z 840.019,A -85,B 0,C 180,E1 -12500.172,E2 -12500.172} C_VEL
LIN {X 0,Y 381.543,Z 829.311,A -85,B 0,C 180,E1 -12501.261,E2 -12501.261} C_VEL
LIN {X 0,Y 382.218,Z 817.402,A -85,B 0,C 180,E1 -12502.208,E2 -12502.208} C_VEL
LIN {X 0,Y 382.633,Z 804.718,A -85,B 0,C 180,E1 -12502.971,E2 -12502.971} C_VEL
LIN {X 0,Y 382.86,Z 791.625,A -85,B 0,C 180,E1 -12503.523,E2 -12503.523} C_VEL
LIN {X 0,Y 382.924,Z 775.649,A -85,B 0,C 180,E1 -12503.911,E2 -12503.911} C_VEL
LIN {X 0,Y 383.511,Z 724.562,A -85,B 0,C 180,E1 -12504.893,E2 -12504.893} C_VEL
LIN {X 0,Y 376.796,Z 708.107,A -85,B 0,C 180,E1 -12505.589,E2 -12505.589} C_VEL
LIN {X 0,Y 376.09,Z 706.197,A -85,B 0,C 180,E1 -12505.748,E2 -12505.748} C_VEL
LIN {X 0,Y 376.022,Z 705.677,A -85,B 0,C 180,E1 -12505.983,E2 -12505.983} C_VEL
LIN {X 0,Y 376.34,Z 705.606,A -85,B 0,C 180,E1 -12507.861,E2 -12507.861} C_VEL
LIN {X 0,Y 376.335,Z 705.606,A -85,B 0,C 180,E1 -12512.142,E2 -12512.142} C_VEL
LIN {X 0,Y 376.197,Z 705.624,A -85,B 0,C 180,E1 -12516.437,E2 -12516.437} C_VEL
LIN {X 0,Y 376.184,Z 705.621,A -85,B 0,C 180,E1 -12517.958,E2 -12517.958} C_VEL
LIN {X 0,Y 375.549,Z 705.706,A -85,B 0,C 180,E1 -12518.852,E2 -12518.852} C_VEL
LIN {X 0,Y 372.621,Z 706.07,A -85,B 0,C 180,E1 -12520.302,E2 -12520.302} C_VEL
LIN {X 0,Y 370.129,Z 706.377,A -85,B 0,C 180,E1 -12521.475,E2 -12521.475} C_VEL
LIN {X 0,Y 369.085,Z 706.51,A -85,B 0,C 180,E1 -12522.385,E2 -12522.385} C_VEL
LIN {X 0,Y 369.017,Z 706.514,A -85,B 0,C 180,E1 -12522.693,E2 -12522.693} C_VEL
LIN {X 0,Y 368.999,Z 706.514,A -85,B 0,C 180,E1 -12525.466,E2 -12525.466} C_VEL
LIN {X 0,Y 368.929,Z 706.521,A -85,B 0,C 180,E1 -12528.897,E2 -12528.897} C_VEL
LIN {X 0,Y 368.902,Z 706.53,A -85,B 0,C 180,E1 -12532.399,E2 -12532.399} C_VEL
LIN {X 0,Y 368.924,Z 706.514,A -85,B 0,C 180,E1 -12535.987,E2 -12535.987} C_VEL
LIN {X 0,Y 368.898,Z 706.532,A -85,B 0,C 180,E1 -12539.693,E2 -12539.693} C_VEL
LIN {X 0,Y 368.901,Z 706.514,A -85,B 0,C 180,E1 -12543.539,E2 -12543.539} C_VEL
LIN {X 0,Y 368.901,Z 706.518,A -85,B 0,C 180,E1 -12546.855,E2 -12546.855} C_VEL
LIN {X 0,Y 368.89,Z 706.531,A -85,B 0,C 180,E1 -12550.375,E2 -12550.375} C_VEL
LIN {X 0,Y 368.861,Z 706.541,A -85,B 0,C 180,E1 -12553.612,E2 -12553.612} C_VEL
LIN {X 0,Y 368.888,Z 706.532,A -85,B 0,C 180,E1 -12556.696,E2 -12556.696} C_VEL
LIN {X 0,Y 368.891,Z 706.537,A -85,B 0,C 180,E1 -12559.649,E2 -12559.649} C_VEL
LIN {X 0,Y 368.899,Z 706.533,A -85,B 0,C 180,E1 -12563.147,E2 -12563.147} C_VEL
LIN {X 0,Y 368.975,Z 706.71,A -85,B 0,C 180,E1 -12566.682,E2 -12566.682} C_VEL
LIN {X 0,Y 369.17,Z 707.601,A -85,B 0,C 180,E1 -12566.849,E2 -12566.849} C_VEL
LIN {X 0,Y 375.35,Z 725.077,A -85,B 0,C 180,E1 -12567.552,E2 -12567.552} C_VEL
LIN {X 0,Y 374.284,Z 782.982,A -85,B 0,C 180,E1 -12568.871,E2 -12568.871} C_VEL
LIN {X 0,Y 374.105,Z 795.263,A -85,B 0,C 180,E1 -12569.325,E2 -12569.325} C_VEL
LIN {X 0,Y 373.771,Z 806.013,A -85,B 0,C 180,E1 -12569.878,E2 -12569.878} C_VEL
LIN {X 0,Y 373.361,Z 816.479,A -85,B 0,C 180,E1 -12570.575,E2 -12570.575} C_VEL
LIN {X 0,Y 372.908,Z 825.1,A -85,B 0,C 180,E1 -12571.276,E2 -12571.276} C_VEL
LIN {X 0,Y 372.458,Z 833.362,A -85,B 0,C 180,E1 -12572.075,E2 -12572.075} C_VEL
LIN {X 0,Y 371.797,Z 842.775,A -85,B 0,C 180,E1 -12573.172,E2 -12573.172} C_VEL
LIN {X 0,Y 371.351,Z 850.202,A -85,B 0,C 180,E1 -12574.196,E2 -12574.196} C_VEL
LIN {X 0,Y 370.756,Z 858.662,A -85,B 0,C 180,E1 -12575.602,E2 -12575.602} C_VEL
LIN {X 0,Y 370.245,Z 864.805,A -85,B 0,C 180,E1 -12576.804,E2 -12576.804} C_VEL
LIN {X 0,Y 369.787,Z 871.11,A -85,B 0,C 180,E1 -12578.3,E2 -12578.3} C_VEL
LIN {X 0,Y 369.557,Z 875.077,A -85,B 0,C 180,E1 -12579.401,E2 -12579.401} C_VEL
LIN {X 0,Y 369.224,Z 880.02,A -85,B 0,C 180,E1 -12581.12,E2 -12581.12} C_VEL
LIN {X 0,Y 369.019,Z 883.703,A -85,B 0,C 180,E1 -12582.83,E2 -12582.83} C_VEL
LIN {X 0,Y 368.864,Z 886.286,A -85,B 0,C 180,E1 -12584.529,E2 -12584.529} C_VEL
LIN {X 0,Y 368.872,Z 887.945,A -85,B 0,C 180,E1 -12586.338,E2 -12586.338} C_VEL
LIN {X 0,Y 368.958,Z 888.424,A -85,B 0,C 180,E1 -12587.905,E2 -12587.905} C_VEL
LIN {X 0,Y 369.101,Z 888.252,A -85,B 0,C 180,E1 -12589.023,E2 -12589.023} C_VEL
LIN {X 0,Y 369.478,Z 886.518,A -85,B 0,C 180,E1 -12591.247,E2 -12591.247} C_VEL
LIN {X 0,Y 369.836,Z 884.107,A -85,B 0,C 180,E1 -12592.905,E2 -12592.905} C_VEL
LIN {X 0,Y 370.367,Z 880.624,A -85,B 0,C 180,E1 -12594.555,E2 -12594.555} C_VEL
LIN {X 0,Y 370.753,Z 877.775,A -85,B 0,C 180,E1 -12595.651,E2 -12595.651} C_VEL
LIN {X 0,Y 371.496,Z 871.215,A -85,B 0,C 180,E1 -12597.56,E2 -12597.56} C_VEL
LIN {X 0,Y 372.288,Z 865.341,A -85,B 0,C 180,E1 -12598.918,E2 -12598.918} C_VEL
LIN {X 0,Y 372.975,Z 859.142,A -85,B 0,C 180,E1 -12600.126,E2 -12600.126} C_VEL
LIN {X 0,Y 373.77,Z 851.653,A -85,B 0,C 180,E1 -12601.347,E2 -12601.347} C_VEL
LIN {X 0,Y 374.505,Z 843.798,A -85,B 0,C 180,E1 -12602.42,E2 -12602.42} C_VEL
LIN {X 0,Y 375.326,Z 834.274,A -85,B 0,C 180,E1 -12603.489,E2 -12603.489} C_VEL
LIN {X 0,Y 375.929,Z 825.703,A -85,B 0,C 180,E1 -12604.288,E2 -12604.288} C_VEL
LIN {X 0,Y 376.402,Z 816.173,A -85,B 0,C 180,E1 -12605.021,E2 -12605.021} C_VEL
LIN {X 0,Y 376.859,Z 805.656,A -85,B 0,C 180,E1 -12605.652,E2 -12605.652} C_VEL
LIN {X 0,Y 377.156,Z 795.416,A -85,B 0,C 180,E1 -12606.117,E2 -12606.117} C_VEL
LIN {X 0,Y 377.265,Z 782.184,A -85,B 0,C 180,E1 -12606.537,E2 -12606.537} C_VEL
LIN {X 0,Y 378.795,Z 727.327,A -85,B 0,C 180,E1 -12607.898,E2 -12607.898} C_VEL
LIN {X 0,Y 373.399,Z 715.514,A -85,B 0,C 180,E1 -12608.694,E2 -12608.694} C_VEL
LIN {X 0,Y 369.259,Z 707.417,A -85,B 0,C 180,E1 -12609.346,E2 -12609.346} C_VEL
LIN {X 0,Y 369.105,Z 706.582,A -85,B 0,C 180,E1 -12609.587,E2 -12609.587} C_VEL
LIN {X 0,Y 369.045,Z 706.512,A -85,B 0,C 180,E1 -12613.772,E2 -12613.772} C_VEL
LIN {X 0,Y 368.998,Z 706.521,A -85,B 0,C 180,E1 -12617.742,E2 -12617.742} C_VEL
LIN {X 0,Y 368.917,Z 706.531,A -85,B 0,C 180,E1 -12621.22,E2 -12621.22} C_VEL
LIN {X 0,Y 368.945,Z 706.528,A -85,B 0,C 180,E1 -12624.776,E2 -12624.776} C_VEL
LIN {X 0,Y 368.938,Z 706.529,A -85,B 0,C 180,E1 -12628.44,E2 -12628.44} C_VEL
LIN {X 0,Y 368.917,Z 706.531,A -85,B 0,C 180,E1 -12630.987,E2 -12630.987} C_VEL
LIN {X 0,Y 368.943,Z 706.527,A -85,B 0,C 180,E1 -12634.853,E2 -12634.853} C_VEL
LIN {X 0,Y 368.915,Z 706.53,A -85,B 0,C 180,E1 -12638.639,E2 -12638.639} C_VEL
LIN {X 0,Y 368.888,Z 706.535,A -85,B 0,C 180,E1 -12642.009,E2 -12642.009} C_VEL
LIN {X 0,Y 368.886,Z 706.534,A -85,B 0,C 180,E1 -12645.175,E2 -12645.175} C_VEL
LIN {X 0,Y 368.889,Z 706.534,A -85,B 0,C 180,E1 -12648.177,E2 -12648.177} C_VEL
LIN {X 0,Y 368.912,Z 706.531,A -85,B 0,C 180,E1 -12651.359,E2 -12651.359} C_VEL
LIN {X 0,Y 368.959,Z 706.705,A -85,B 0,C 180,E1 -12654.957,E2 -12654.957} C_VEL
LIN {X 0,Y 372.606,Z 722.044,A -85,B 0,C 180,E1 -12658.119,E2 -12658.119} C_VEL
LIN {X 0,Y 374.97,Z 732.819,A -85,B 0,C 180,E1 -12660.217,E2 -12660.217} C_VEL
LIN {X 0,Y 375.031,Z 736.277,A -85,B 0,C 180,E1 -12660.839,E2 -12660.839} C_VEL
LIN {X 0,Y 372.99,Z 758.31,A -85,B 0,C 180,E1 -12664.62,E2 -12664.62} C_VEL
LIN {X 0,Y 371.568,Z 776.463,A -85,B 0,C 180,E1 -12667.661,E2 -12667.661} C_VEL
LIN {X 0,Y 374.051,Z 796.231,A -85,B 0,C 180,E1 -12668.434,E2 -12668.434} C_VEL
LIN {X 0,Y 376.485,Z 827.625,A -85,B 0,C 180,E1 -12669.473,E2 -12669.473} C_VEL
LIN {X 0,Y 375.267,Z 874.9,A -85,B 0,C 180,E1 -12670.583,E2 -12670.583} C_VEL
LIN {X 0,Y 374.846,Z 893.617,A -85,B 0,C 180,E1 -12670.987,E2 -12670.987} C_VEL
LIN {X 0,Y 374.215,Z 906.965,A -85,B 0,C 180,E1 -12671.486,E2 -12671.486} C_VEL
LIN {X 0,Y 373.259,Z 919.585,A -85,B 0,C 180,E1 -12672.182,E2 -12672.182} C_VEL
LIN {X 0,Y 372.101,Z 932.074,A -85,B 0,C 180,E1 -12673.117,E2 -12673.117} C_VEL
LIN {X 0,Y 371.049,Z 943.277,A -85,B 0,C 180,E1 -12674.199,E2 -12674.199} C_VEL
LIN {X 0,Y 370.149,Z 953.401,A -85,B 0,C 180,E1 -12675.428,E2 -12675.428} C_VEL
LIN {X 0,Y 369.432,Z 962.611,A -85,B 0,C 180,E1 -12676.802,E2 -12676.802} C_VEL
LIN {X 0,Y 368.651,Z 971.603,A -85,B 0,C 180,E1 -12678.451,E2 -12678.451} C_VEL
LIN {X 0,Y 368.228,Z 978.838,A -85,B 0,C 180,E1 -12680.107,E2 -12680.107} C_VEL
LIN {X 0,Y 368.076,Z 984.637,A -85,B 0,C 180,E1 -12681.765,E2 -12681.765} C_VEL
LIN {X 0,Y 368.059,Z 989.203,A -85,B 0,C 180,E1 -12683.42,E2 -12683.42} C_VEL
LIN {X 0,Y 368.099,Z 991.613,A -85,B 0,C 180,E1 -12684.52,E2 -12684.52} C_VEL
LIN {X 0,Y 368.251,Z 993.588,A -85,B 0,C 180,E1 -12685.62,E2 -12685.62} C_VEL
LIN {X 0,Y 368.288,Z 995.084,A -85,B 0,C 180,E1 -12686.716,E2 -12686.716} C_VEL
LIN {X 0,Y 368.325,Z 996.126,A -85,B 0,C 180,E1 -12687.811,E2 -12687.811} C_VEL
LIN {X 0,Y 368.38,Z 996.761,A -85,B 0,C 180,E1 -12688.905,E2 -12688.905} C_VEL
LIN {X 0,Y 368.428,Z 996.988,A -85,B 0,C 180,E1 -12689.998,E2 -12689.998} C_VEL
LIN {X 0,Y 368.378,Z 996.771,A -85,B 0,C 180,E1 -12691.092,E2 -12691.092} C_VEL
LIN {X 0,Y 368.322,Z 996.115,A -85,B 0,C 180,E1 -12692.185,E2 -12692.185} C_VEL
LIN {X 0,Y 368.284,Z 995.056,A -85,B 0,C 180,E1 -12693.28,E2 -12693.28} C_VEL
LIN {X 0,Y 368.243,Z 993.582,A -85,B 0,C 180,E1 -12694.377,E2 -12694.377} C_VEL
LIN {X 0,Y 368.09,Z 990.486,A -85,B 0,C 180,E1 -12696.026,E2 -12696.026} C_VEL
LIN {X 0,Y 368.054,Z 986.334,A -85,B 0,C 180,E1 -12697.68,E2 -12697.68} C_VEL
LIN {X 0,Y 368.162,Z 980.01,A -85,B 0,C 180,E1 -12699.614,E2 -12699.614} C_VEL
LIN {X 0,Y 368.536,Z 973.133,A -85,B 0,C 180,E1 -12701.27,E2 -12701.27} C_VEL
LIN {X 0,Y 369.19,Z 964.654,A -85,B 0,C 180,E1 -12702.923,E2 -12702.923} C_VEL
LIN {X 0,Y 369.975,Z 955.664,A -85,B 0,C 180,E1 -12704.352,E2 -12704.352} C_VEL
LIN {X 0,Y 370.855,Z 945.492,A -85,B 0,C 180,E1 -12705.665,E2 -12705.665} C_VEL
LIN {X 0,Y 372.214,Z 933.704,A -85,B 0,C 180,E1 -12706.874,E2 -12706.874} C_VEL
LIN {X 0,Y 373.253,Z 922.078,A -85,B 0,C 180,E1 -12707.815,E2 -12707.815} C_VEL
LIN {X 0,Y 374.417,Z 908.815,A -85,B 0,C 180,E1 -12708.607,E2 -12708.607} C_VEL
LIN {X 0,Y 375.226,Z 895.476,A -85,B 0,C 180,E1 -12709.168,E2 -12709.168} C_VEL
LIN {X 0,Y 375.643,Z 880.689,A -85,B 0,C 180,E1 -12709.536,E2 -12709.536} C_VEL
LIN {X 0,Y 376.42,Z 825.262,A -85,B 0,C 180,E1 -12710.622,E2 -12710.622} C_VEL
LIN {X 0,Y 372.821,Z 790.508,A -85,B 0,C 180,E1 -12711.553,E2 -12711.553} C_VEL
LIN {X 0,Y 371.349,Z 778.539,A -85,B 0,C 180,E1 -12711.935,E2 -12711.935} C_VEL
LIN {X 0,Y 373.041,Z 758.22,A -85,B 0,C 180,E1 -12715.378,E2 -12715.378} C_VEL
LIN {X 0,Y 375.049,Z 736.506,A -85,B 0,C 180,E1 -12719.155,E2 -12719.155} C_VEL
LIN {X 0,Y 375.052,Z 733.133,A -85,B 0,C 180,E1 -12719.772,E2 -12719.772} C_VEL
LIN {X 0,Y 372.473,Z 721.034,A -85,B 0,C 180,E1 -12722.208,E2 -12722.208} C_VEL
LIN {X 0,Y 369.193,Z 707.737,A -85,B 0,C 180,E1 -12725.06,E2 -12725.06} C_VEL
LIN {X 0,Y 368.954,Z 706.596,A -85,B 0,C 180,E1 -12725.388,E2 -12725.388} C_VEL
LIN {X 0,Y 368.896,Z 706.535,A -85,B 0,C 180,E1 -12728.952,E2 -12728.952} C_VEL
LIN {X 0,Y 368.874,Z 706.538,A -85,B 0,C 180,E1 -12732.008,E2 -12732.008} C_VEL
LIN {X 0,Y 368.878,Z 706.533,A -85,B 0,C 180,E1 -12735.175,E2 -12735.175} C_VEL
LIN {X 0,Y 368.875,Z 706.537,A -85,B 0,C 180,E1 -12738.176,E2 -12738.176} C_VEL
LIN {X 0,Y 368.901,Z 706.531,A -85,B 0,C 180,E1 -12741.358,E2 -12741.358} C_VEL
LIN {X 0,Y 368.927,Z 706.517,A -85,B 0,C 180,E1 -12745.145,E2 -12745.145} C_VEL
LIN {X 0,Y 368.918,Z 706.529,A -85,B 0,C 180,E1 -12749.046,E2 -12749.046} C_VEL
LIN {X 0,Y 368.976,Z 706.521,A -85,B 0,C 180,E1 -12751.564,E2 -12751.564} C_VEL
LIN {X 0,Y 368.946,Z 706.524,A -85,B 0,C 180,E1 -12755.224,E2 -12755.224} C_VEL
LIN {X 0,Y 368.926,Z 706.523,A -85,B 0,C 180,E1 -12758.973,E2 -12758.973} C_VEL
LIN {X 0,Y 368.979,Z 706.515,A -85,B 0,C 180,E1 -12762.257,E2 -12762.257} C_VEL
LIN {X 0,Y 369.004,Z 706.519,A -85,B 0,C 180,E1 -12765.665,E2 -12765.665} C_VEL
LIN {X 0,Y 369.01,Z 706.517,A -85,B 0,C 180,E1 -12769.021,E2 -12769.021} C_VEL
LIN {X 0,Y 369.149,Z 706.501,A -85,B 0,C 180,E1 -12772.342,E2 -12772.342} C_VEL
LIN {X 0,Y 369.13,Z 706.5,A -85,B 0,C 180,E1 -12774.538,E2 -12774.538} C_VEL
LIN {X 0,Y 369.307,Z 706.481,A -85,B 0,C 180,E1 -12777.819,E2 -12777.819} C_VEL
LIN {X 0,Y 369.446,Z 706.459,A -85,B 0,C 180,E1 -12780,E2 -12780} C_VEL
LIN {X 0,Y 369.306,Z 706.482,A -85,B 0,C 180,E1 -12782.181,E2 -12782.181} C_VEL
LIN {X 0,Y 369.186,Z 706.498,A -85,B 0,C 180,E1 -12786.671,E2 -12786.671} C_VEL
LIN {X 0,Y 369.126,Z 706.5,A -85,B 0,C 180,E1 -12788.761,E2 -12788.761} C_VEL
LIN {X 0,Y 368.994,Z 706.517,A -85,B 0,C 180,E1 -12792.094,E2 -12792.094} C_VEL
LIN {X 0,Y 368.986,Z 706.516,A -85,B 0,C 180,E1 -12795.466,E2 -12795.466} C_VEL
LIN {X 0,Y 368.946,Z 706.526,A -85,B 0,C 180,E1 -12798.895,E2 -12798.895} C_VEL
LIN {X 0,Y 368.911,Z 706.525,A -85,B 0,C 180,E1 -12802.397,E2 -12802.397} C_VEL
LIN {X 0,Y 368.989,Z 706.523,A -85,B 0,C 180,E1 -12805.981,E2 -12805.981} C_VEL
LIN {X 0,Y 368.905,Z 706.529,A -85,B 0,C 180,E1 -12809.692,E2 -12809.692} C_VEL
LIN {X 0,Y 368.889,Z 706.525,A -85,B 0,C 180,E1 -12813.045,E2 -12813.045} C_VEL
LIN {X 0,Y 368.91,Z 706.526,A -85,B 0,C 180,E1 -12816.198,E2 -12816.198} C_VEL
LIN {X 0,Y 368.897,Z 706.528,A -85,B 0,C 180,E1 -12818.954,E2 -12818.954} C_VEL
LIN {X 0,Y 368.907,Z 706.531,A -85,B 0,C 180,E1 -12822.606,E2 -12822.606} C_VEL
LIN {X 0,Y 368.981,Z 706.817,A -85,B 0,C 180,E1 -12823.351,E2 -12823.351} C_VEL
LIN {X 0,Y 369.322,Z 708.089,A -85,B 0,C 180,E1 -12823.522,E2 -12823.522} C_VEL
LIN {X 0,Y 377.717,Z 727.412,A -85,B 0,C 180,E1 -12824.497,E2 -12824.497} C_VEL
LIN {X 0,Y 377.06,Z 788.003,A -85,B 0,C 180,E1 -12825.729,E2 -12825.729} C_VEL
LIN {X 0,Y 376.932,Z 801.015,A -85,B 0,C 180,E1 -12826.175,E2 -12826.175} C_VEL
LIN {X 0,Y 376.607,Z 813.745,A -85,B 0,C 180,E1 -12826.846,E2 -12826.846} C_VEL
LIN {X 0,Y 376.037,Z 825.937,A -85,B 0,C 180,E1 -12827.717,E2 -12827.717} C_VEL
LIN {X 0,Y 375.322,Z 836.071,A -85,B 0,C 180,E1 -12828.643,E2 -12828.643} C_VEL
LIN {X 0,Y 374.463,Z 846.387,A -85,B 0,C 180,E1 -12829.825,E2 -12829.825} C_VEL
LIN {X 0,Y 373.44,Z 856.493,A -85,B 0,C 180,E1 -12831.265,E2 -12831.265} C_VEL
LIN {X 0,Y 372.654,Z 863.526,A -85,B 0,C 180,E1 -12832.492,E2 -12832.492} C_VEL
LIN {X 0,Y 371.795,Z 871.222,A -85,B 0,C 180,E1 -12834.129,E2 -12834.129} C_VEL
LIN {X 0,Y 371.075,Z 877.143,A -85,B 0,C 180,E1 -12835.708,E2 -12835.708} C_VEL
LIN {X 0,Y 370.423,Z 881.828,A -85,B 0,C 180,E1 -12837.269,E2 -12837.269} C_VEL
LIN {X 0,Y 369.899,Z 886.05,A -85,B 0,C 180,E1 -12839.139,E2 -12839.139} C_VEL
LIN {X 0,Y 369.491,Z 889.02,A -85,B 0,C 180,E1 -12841.041,E2 -12841.041} C_VEL
LIN {X 0,Y 369.197,Z 891.009,A -85,B 0,C 180,E1 -12843.469,E2 -12843.469} C_VEL
LIN {X 0,Y 369.072,Z 891.242,A -85,B 0,C 180,E1 -12845.235,E2 -12845.235} C_VEL
LIN {X 0,Y 369.069,Z 890.824,A -85,B 0,C 180,E1 -12846.431,E2 -12846.431} C_VEL
LIN {X 0,Y 369.151,Z 889.952,A -85,B 0,C 180,E1 -12847.621,E2 -12847.621} C_VEL
LIN {X 0,Y 369.315,Z 888.55,A -85,B 0,C 180,E1 -12848.823,E2 -12848.823} C_VEL
LIN {X 0,Y 369.634,Z 885.659,A -85,B 0,C 180,E1 -12850.567,E2 -12850.567} C_VEL
LIN {X 0,Y 370.069,Z 881.629,A -85,B 0,C 180,E1 -12852.312,E2 -12852.312} C_VEL
LIN {X 0,Y 370.629,Z 876.387,A -85,B 0,C 180,E1 -12854.043,E2 -12854.043} C_VEL
LIN {X 0,Y 371.305,Z 869.759,A -85,B 0,C 180,E1 -12855.757,E2 -12855.757} C_VEL
LIN {X 0,Y 372.217,Z 861.404,A -85,B 0,C 180,E1 -12857.461,E2 -12857.461} C_VEL
LIN {X 0,Y 373.041,Z 852.234,A -85,B 0,C 180,E1 -12858.971,E2 -12858.971} C_VEL
LIN {X 0,Y 373.866,Z 842.455,A -85,B 0,C 180,E1 -12860.261,E2 -12860.261} C_VEL
LIN {X 0,Y 374.61,Z 832.08,A -85,B 0,C 180,E1 -12861.37,E2 -12861.37} C_VEL
LIN {X 0,Y 375.328,Z 820.714,A -85,B 0,C 180,E1 -12862.335,E2 -12862.335} C_VEL
LIN {X 0,Y 375.813,Z 808.709,A -85,B 0,C 180,E1 -12863.12,E2 -12863.12} C_VEL
LIN {X 0,Y 376.087,Z 795.232,A -85,B 0,C 180,E1 -12863.746,E2 -12863.746} C_VEL
LIN {X 0,Y 376.201,Z 782.22,A -85,B 0,C 180,E1 -12864.124,E2 -12864.124} C_VEL
LIN {X 0,Y 376.83,Z 726.169,A -85,B 0,C 180,E1 -12865.225,E2 -12865.225} C_VEL
LIN {X 0,Y 369.715,Z 708.916,A -85,B 0,C 180,E1 -12865.982,E2 -12865.982} C_VEL
LIN {X 0,Y 369.066,Z 707.007,A -85,B 0,C 180,E1 -12866.146,E2 -12866.146} C_VEL
LIN {X 0,Y 369.053,Z 706.516,A -85,B 0,C 180,E1 -12866.453,E2 -12866.453} C_VEL
LIN {X 0,Y 369.304,Z 706.483,A -85,B 0,C 180,E1 -12867.82,E2 -12867.82} C_VEL
LIN {X 0,Y 369.298,Z 706.482,A -85,B 0,C 180,E1 -12872.183,E2 -12872.183} C_VEL
LIN {X 0,Y 369.159,Z 706.499,A -85,B 0,C 180,E1 -12876.561,E2 -12876.561} C_VEL
LIN {X 0,Y 369.061,Z 706.512,A -85,B 0,C 180,E1 -12879.87,E2 -12879.87} C_VEL
LIN {X 0,Y 369.017,Z 706.514,A -85,B 0,C 180,E1 -12882.693,E2 -12882.693} C_VEL
LIN {X 0,Y 368.384,Z 706.595,A -85,B 0,C 180,E1 -12883.604,E2 -12883.604} C_VEL
LIN {X 0,Y 365.509,Z 706.956,A -85,B 0,C 180,E1 -12885.085,E2 -12885.085} C_VEL
LIN {X 0,Y 363.05,Z 707.263,A -85,B 0,C 180,E1 -12886.283,E2 -12886.283} C_VEL
LIN {X 0,Y 361.997,Z 707.393,A -85,B 0,C 180,E1 -12887.211,E2 -12887.211} C_VEL
LIN {X 0,Y 361.914,Z 707.401,A -85,B 0,C 180,E1 -12887.525,E2 -12887.525} C_VEL
LIN {X 0,Y 361.87,Z 707.403,A -85,B 0,C 180,E1 -12891.215,E2 -12891.215} C_VEL
LIN {X 0,Y 361.867,Z 707.406,A -85,B 0,C 180,E1 -12894.102,E2 -12894.102} C_VEL
LIN {X 0,Y 361.84,Z 707.403,A -85,B 0,C 180,E1 -12897.786,E2 -12897.786} C_VEL
LIN {X 0,Y 361.833,Z 707.413,A -85,B 0,C 180,E1 -12901.281,E2 -12901.281} C_VEL
LIN {X 0,Y 361.857,Z 707.387,A -85,B 0,C 180,E1 -12904.282,E2 -12904.282} C_VEL
LIN {X 0,Y 361.862,Z 707.398,A -85,B 0,C 180,E1 -12907.222,E2 -12907.222} C_VEL
LIN {X 0,Y 361.815,Z 707.413,A -85,B 0,C 180,E1 -12910.751,E2 -12910.751} C_VEL
LIN {X 0,Y 361.802,Z 707.415,A -85,B 0,C 180,E1 -12914.373,E2 -12914.373} C_VEL
LIN {X 0,Y 361.829,Z 707.415,A -85,B 0,C 180,E1 -12917.571,E2 -12917.571} C_VEL
LIN {X 0,Y 361.847,Z 707.412,A -85,B 0,C 180,E1 -12921.572,E2 -12921.572} C_VEL
LIN {X 0,Y 361.874,Z 707.409,A -85,B 0,C 180,E1 -12924.657,E2 -12924.657} C_VEL
LIN {X 0,Y 361.958,Z 707.644,A -85,B 0,C 180,E1 -12926.394,E2 -12926.394} C_VEL
LIN {X 0,Y 362.206,Z 708.647,A -85,B 0,C 180,E1 -12926.55,E2 -12926.55} C_VEL
LIN {X 0,Y 368.39,Z 726.141,A -85,B 0,C 180,E1 -12927.27,E2 -12927.27} C_VEL
LIN {X 0,Y 367.385,Z 784.095,A -85,B 0,C 180,E1 -12928.627,E2 -12928.627} C_VEL
LIN {X 0,Y 367.209,Z 796.243,A -85,B 0,C 180,E1 -12929.087,E2 -12929.087} C_VEL
LIN {X 0,Y 366.921,Z 806.012,A -85,B 0,C 180,E1 -12929.59,E2 -12929.59} C_VEL
LIN {X 0,Y 366.528,Z 816.084,A -85,B 0,C 180,E1 -12930.255,E2 -12930.255} C_VEL
LIN {X 0,Y 365.912,Z 826.848,A -85,B 0,C 180,E1 -12931.146,E2 -12931.146} C_VEL
LIN {X 0,Y 365.467,Z 835.196,A -85,B 0,C 180,E1 -12931.985,E2 -12931.985} C_VEL
LIN {X 0,Y 364.808,Z 844.322,A -85,B 0,C 180,E1 -12933.081,E2 -12933.081} C_VEL
LIN {X 0,Y 364.291,Z 852.588,A -85,B 0,C 180,E1 -12934.273,E2 -12934.273} C_VEL
LIN {X 0,Y 363.737,Z 860.203,A -85,B 0,C 180,E1 -12935.581,E2 -12935.581} C_VEL
LIN {X 0,Y 363.18,Z 866.793,A -85,B 0,C 180,E1 -12936.929,E2 -12936.929} C_VEL
LIN {X 0,Y 362.767,Z 872.75,A -85,B 0,C 180,E1 -12938.402,E2 -12938.402} C_VEL
LIN {X 0,Y 362.474,Z 876.787,A -85,B 0,C 180,E1 -12939.573,E2 -12939.573} C_VEL
LIN {X 0,Y 362.169,Z 881.557,A -85,B 0,C 180,E1 -12941.325,E2 -12941.325} C_VEL
LIN {X 0,Y 361.942,Z 885.12,A -85,B 0,C 180,E1 -12943.066,E2 -12943.066} C_VEL
LIN {X 0,Y 361.867,Z 886.968,A -85,B 0,C 180,E1 -12944.222,E2 -12944.222} C_VEL
LIN {X 0,Y 361.885,Z 889.088,A -85,B 0,C 180,E1 -12946.523,E2 -12946.523} C_VEL
LIN {X 0,Y 361.925,Z 889.507,A -85,B 0,C 180,E1 -12947.666,E2 -12947.666} C_VEL
LIN {X 0,Y 362.073,Z 889.437,A -85,B 0,C 180,E1 -12948.807,E2 -12948.807} C_VEL
LIN {X 0,Y 362.458,Z 888.056,A -85,B 0,C 180,E1 -12951.076,E2 -12951.076} C_VEL
LIN {X 0,Y 362.698,Z 886.635,A -85,B 0,C 180,E1 -12952.204,E2 -12952.204} C_VEL
LIN {X 0,Y 363.396,Z 882.573,A -85,B 0,C 180,E1 -12954.451,E2 -12954.451} C_VEL
LIN {X 0,Y 363.99,Z 878.183,A -85,B 0,C 180,E1 -12956.125,E2 -12956.125} C_VEL
LIN {X 0,Y 364.699,Z 872.56,A -85,B 0,C 180,E1 -12957.791,E2 -12957.791} C_VEL
LIN {X 0,Y 365.504,Z 866.907,A -85,B 0,C 180,E1 -12959.143,E2 -12959.143} C_VEL
LIN {X 0,Y 366.235,Z 861.163,A -85,B 0,C 180,E1 -12960.307,E2 -12960.307} C_VEL
LIN {X 0,Y 367.119,Z 853.172,A -85,B 0,C 180,E1 -12961.645,E2 -12961.645} C_VEL
LIN {X 0,Y 368.007,Z 844.24,A -85,B 0,C 180,E1 -12962.873,E2 -12962.873} C_VEL
LIN {X 0,Y 368.761,Z 835.91,A -85,B 0,C 180,E1 -12963.825,E2 -12963.825} C_VEL
LIN {X 0,Y 369.392,Z 827.431,A -85,B 0,C 180,E1 -12964.638,E2 -12964.638} C_VEL
LIN {X 0,Y 369.969,Z 817.085,A -85,B 0,C 180,E1 -12965.45,E2 -12965.45} C_VEL
LIN {X 0,Y 370.456,Z 806.593,A -85,B 0,C 180,E1 -12966.092,E2 -12966.092} C_VEL
LIN {X 0,Y 370.771,Z 795.878,A -85,B 0,C 180,E1 -12966.584,E2 -12966.584} C_VEL
LIN {X 0,Y 370.903,Z 782.669,A -85,B 0,C 180,E1 -12967.009,E2 -12967.009} C_VEL
LIN {X 0,Y 372.584,Z 729.396,A -85,B 0,C 180,E1 -12968.362,E2 -12968.362} C_VEL
LIN {X 0,Y 367.002,Z 717.508,A -85,B 0,C 180,E1 -12969.228,E2 -12969.228} C_VEL
LIN {X 0,Y 363.142,Z 710.388,A -85,B 0,C 180,E1 -12969.833,E2 -12969.833} C_VEL
LIN {X 0,Y 362.118,Z 708.032,A -85,B 0,C 180,E1 -12970.059,E2 -12970.059} C_VEL
LIN {X 0,Y 361.995,Z 707.429,A -85,B 0,C 180,E1 -12970.345,E2 -12970.345} C_VEL
LIN {X 0,Y 362.006,Z 707.389,A -85,B 0,C 180,E1 -12973.898,E2 -12973.898} C_VEL
LIN {X 0,Y 361.936,Z 707.403,A -85,B 0,C 180,E1 -12976.934,E2 -12976.934} C_VEL
LIN {X 0,Y 361.894,Z 707.406,A -85,B 0,C 180,E1 -12980.46,E2 -12980.46} C_VEL
LIN {X 0,Y 361.901,Z 707.405,A -85,B 0,C 180,E1 -12984.112,E2 -12984.112} C_VEL
LIN {X 0,Y 361.871,Z 707.409,A -85,B 0,C 180,E1 -12987.782,E2 -12987.782} C_VEL
LIN {X 0,Y 361.854,Z 707.413,A -85,B 0,C 180,E1 -12991.285,E2 -12991.285} C_VEL
LIN {X 0,Y 361.861,Z 707.409,A -85,B 0,C 180,E1 -12994.28,E2 -12994.28} C_VEL
LIN {X 0,Y 361.87,Z 707.409,A -85,B 0,C 180,E1 -12997.222,E2 -12997.222} C_VEL
LIN {X 0,Y 361.842,Z 707.411,A -85,B 0,C 180,E1 -13000.755,E2 -13000.755} C_VEL
LIN {X 0,Y 361.824,Z 707.414,A -85,B 0,C 180,E1 -13004.368,E2 -13004.368} C_VEL
LIN {X 0,Y 361.842,Z 707.413,A -85,B 0,C 180,E1 -13007.567,E2 -13007.567} C_VEL
LIN {X 0,Y 361.873,Z 707.406,A -85,B 0,C 180,E1 -13010.973,E2 -13010.973} C_VEL
LIN {X 0,Y 361.917,Z 707.616,A -85,B 0,C 180,E1 -13014.584,E2 -13014.584} C_VEL
LIN {X 0,Y 365.545,Z 722.736,A -85,B 0,C 180,E1 -13017.774,E2 -13017.774} C_VEL
LIN {X 0,Y 367.987,Z 733.892,A -85,B 0,C 180,E1 -13019.996,E2 -13019.996} C_VEL
LIN {X 0,Y 368.196,Z 736.913,A -85,B 0,C 180,E1 -13020.559,E2 -13020.559} C_VEL
LIN {X 0,Y 365.95,Z 760.163,A -85,B 0,C 180,E1 -13024.629,E2 -13024.629} C_VEL
LIN {X 0,Y 364.775,Z 774.146,A -85,B 0,C 180,E1 -13027.009,E2 -13027.009} C_VEL
LIN {X 0,Y 367.729,Z 797.456,A -85,B 0,C 180,E1 -13027.975,E2 -13027.975} C_VEL
LIN {X 0,Y 370.047,Z 828.166,A -85,B 0,C 180,E1 -13029.018,E2 -13029.018} C_VEL
LIN {X 0,Y 368.024,Z 894.139,A -85,B 0,C 180,E1 -13030.693,E2 -13030.693} C_VEL
LIN {X 0,Y 367.421,Z 906.22,A -85,B 0,C 180,E1 -13031.167,E2 -13031.167} C_VEL
LIN {X 0,Y 366.47,Z 918.267,A -85,B 0,C 180,E1 -13031.841,E2 -13031.841} C_VEL
LIN {X 0,Y 365.301,Z 930.826,A -85,B 0,C 180,E1 -13032.793,E2 -13032.793} C_VEL
LIN {X 0,Y 364.174,Z 942.081,A -85,B 0,C 180,E1 -13033.892,E2 -13033.892} C_VEL
LIN {X 0,Y 363.231,Z 952.251,A -85,B 0,C 180,E1 -13035.144,E2 -13035.144} C_VEL
LIN {X 0,Y 362.586,Z 960.136,A -85,B 0,C 180,E1 -13036.316,E2 -13036.316} C_VEL
LIN {X 0,Y 361.726,Z 969.109,A -85,B 0,C 180,E1 -13037.943,E2 -13037.943} C_VEL
LIN {X 0,Y 361.222,Z 976.632,A -85,B 0,C 180,E1 -13039.63,E2 -13039.63} C_VEL
LIN {X 0,Y 361,Z 983.568,A -85,B 0,C 180,E1 -13041.603,E2 -13041.603} C_VEL
LIN {X 0,Y 361.01,Z 988.154,A -85,B 0,C 180,E1 -13043.291,E2 -13043.291} C_VEL
LIN {X 0,Y 361.033,Z 990.567,A -85,B 0,C 180,E1 -13044.413,E2 -13044.413} C_VEL
LIN {X 0,Y 361.185,Z 992.548,A -85,B 0,C 180,E1 -13045.534,E2 -13045.534} C_VEL
LIN {X 0,Y 361.243,Z 994.059,A -85,B 0,C 180,E1 -13046.652,E2 -13046.652} C_VEL
LIN {X 0,Y 361.286,Z 995.106,A -85,B 0,C 180,E1 -13047.769,E2 -13047.769} C_VEL
LIN {X 0,Y 361.346,Z 995.745,A -85,B 0,C 180,E1 -13048.884,E2 -13048.884} C_VEL
LIN {X 0,Y 361.4,Z 995.977,A -85,B 0,C 180,E1 -13049.998,E2 -13049.998} C_VEL
LIN {X 0,Y 361.343,Z 995.767,A -85,B 0,C 180,E1 -13051.113,E2 -13051.113} C_VEL
LIN {X 0,Y 361.28,Z 995.113,A -85,B 0,C 180,E1 -13052.228,E2 -13052.228} C_VEL
LIN {X 0,Y 361.239,Z 994.054,A -85,B 0,C 180,E1 -13053.344,E2 -13053.344} C_VEL
LIN {X 0,Y 361.179,Z 992.578,A -85,B 0,C 180,E1 -13054.462,E2 -13054.462} C_VEL
LIN {X 0,Y 361.035,Z 989.488,A -85,B 0,C 180,E1 -13056.144,E2 -13056.144} C_VEL
LIN {X 0,Y 360.995,Z 985.339,A -85,B 0,C 180,E1 -13057.831,E2 -13057.831} C_VEL
LIN {X 0,Y 361.114,Z 979.027,A -85,B 0,C 180,E1 -13059.803,E2 -13059.803} C_VEL
LIN {X 0,Y 361.518,Z 972.167,A -85,B 0,C 180,E1 -13061.492,E2 -13061.492} C_VEL
LIN {X 0,Y 362.251,Z 963.716,A -85,B 0,C 180,E1 -13063.175,E2 -13063.175} C_VEL
LIN {X 0,Y 363.007,Z 955.122,A -85,B 0,C 180,E1 -13064.576,E2 -13064.576} C_VEL
LIN {X 0,Y 364.036,Z 944.625,A -85,B 0,C 180,E1 -13065.967,E2 -13065.967} C_VEL
LIN {X 0,Y 365.354,Z 932.862,A -85,B 0,C 180,E1 -13067.201,E2 -13067.201} C_VEL
LIN {X 0,Y 366.493,Z 921.308,A -85,B 0,C 180,E1 -13068.155,E2 -13068.155} C_VEL
LIN {X 0,Y 367.583,Z 909.464,A -85,B 0,C 180,E1 -13068.893,E2 -13068.893} C_VEL
LIN {X 0,Y 368.471,Z 895.898,A -85,B 0,C 180,E1 -13069.497,E2 -13069.497} C_VEL
LIN {X 0,Y 368.972,Z 882.485,A -85,B 0,C 180,E1 -13069.868,E2 -13069.868} C_VEL
LIN {X 0,Y 369.863,Z 826.564,A -85,B 0,C 180,E1 -13070.98,E2 -13070.98} C_VEL
LIN {X 0,Y 366.34,Z 792.147,A -85,B 0,C 180,E1 -13071.928,E2 -13071.928} C_VEL
LIN {X 0,Y 364.514,Z 777.81,A -85,B 0,C 180,E1 -13072.37,E2 -13072.37} C_VEL
LIN {X 0,Y 364.931,Z 772.363,A -85,B 0,C 180,E1 -13073.251,E2 -13073.251} C_VEL
LIN {X 0,Y 366.546,Z 754.01,A -85,B 0,C 180,E1 -13076.472,E2 -13076.472} C_VEL
LIN {X 0,Y 368.25,Z 737.363,A -85,B 0,C 180,E1 -13079.433,E2 -13079.433} C_VEL
LIN {X 0,Y 367.886,Z 733.147,A -85,B 0,C 180,E1 -13080.247,E2 -13080.247} C_VEL
LIN {X 0,Y 365.025,Z 720.206,A -85,B 0,C 180,E1 -13082.943,E2 -13082.943} C_VEL
LIN {X 0,Y 362.019,Z 708.178,A -85,B 0,C 180,E1 -13085.617,E2 -13085.617} C_VEL
LIN {X 0,Y 361.881,Z 707.452,A -85,B 0,C 180,E1 -13085.89,E2 -13085.89} C_VEL
LIN {X 0,Y 361.862,Z 707.412,A -85,B 0,C 180,E1 -13089.025,E2 -13089.025} C_VEL
LIN {X 0,Y 361.828,Z 707.409,A -85,B 0,C 180,E1 -13092.827,E2 -13092.827} C_VEL
LIN {X 0,Y 361.813,Z 707.409,A -85,B 0,C 180,E1 -13095.945,E2 -13095.945} C_VEL
LIN {X 0,Y 361.827,Z 707.406,A -85,B 0,C 180,E1 -13099.243,E2 -13099.243} C_VEL
LIN {X 0,Y 361.862,Z 707.411,A -85,B 0,C 180,E1 -13102.774,E2 -13102.774} C_VEL
LIN {X 0,Y 361.845,Z 707.405,A -85,B 0,C 180,E1 -13105.719,E2 -13105.719} C_VEL
LIN {X 0,Y 361.866,Z 707.411,A -85,B 0,C 180,E1 -13109.671,E2 -13109.671} C_VEL
LIN {X 0,Y 361.944,Z 707.402,A -85,B 0,C 180,E1 -13113.474,E2 -13113.474} C_VEL
LIN {X 0,Y 361.879,Z 707.408,A -85,B 0,C 180,E1 -13117.144,E2 -13117.144} C_VEL
LIN {X 0,Y 361.909,Z 707.402,A -85,B 0,C 180,E1 -13120.724,E2 -13120.724} C_VEL
LIN {X 0,Y 361.936,Z 707.401,A -85,B 0,C 180,E1 -13124.226,E2 -13124.226} C_VEL
LIN {X 0,Y 361.987,Z 707.385,A -85,B 0,C 180,E1 -13126.527,E2 -13126.527} C_VEL
LIN {X 0,Y 362.019,Z 707.387,A -85,B 0,C 180,E1 -13129.938,E2 -13129.938} C_VEL
LIN {X 0,Y 362.148,Z 707.372,A -85,B 0,C 180,E1 -13133.314,E2 -13133.314} C_VEL
LIN {X 0,Y 362.271,Z 707.357,A -85,B 0,C 180,E1 -13137.777,E2 -13137.777} C_VEL
LIN {X 0,Y 362.415,Z 707.334,A -85,B 0,C 180,E1 -13140,E2 -13140} C_VEL
LIN {X 0,Y 362.27,Z 707.359,A -85,B 0,C 180,E1 -13142.224,E2 -13142.224} C_VEL
LIN {X 0,Y 362.159,Z 707.375,A -85,B 0,C 180,E1 -13146.687,E2 -13146.687} C_VEL
LIN {X 0,Y 362.062,Z 707.38,A -85,B 0,C 180,E1 -13148.934,E2 -13148.934} C_VEL
LIN {X 0,Y 361.949,Z 707.394,A -85,B 0,C 180,E1 -13152.333,E2 -13152.333} C_VEL
LIN {X 0,Y 361.95,Z 707.401,A -85,B 0,C 180,E1 -13154.621,E2 -13154.621} C_VEL
LIN {X 0,Y 361.945,Z 707.398,A -85,B 0,C 180,E1 -13158.1,E2 -13158.1} C_VEL
LIN {X 0,Y 361.85,Z 707.407,A -85,B 0,C 180,E1 -13161.656,E2 -13161.656} C_VEL
LIN {X 0,Y 361.915,Z 707.4,A -85,B 0,C 180,E1 -13165.291,E2 -13165.291} C_VEL
LIN {X 0,Y 361.898,Z 707.396,A -85,B 0,C 180,E1 -13167.78,E2 -13167.78} C_VEL
LIN {X 0,Y 361.828,Z 707.411,A -85,B 0,C 180,E1 -13171.631,E2 -13171.631} C_VEL
LIN {X 0,Y 361.866,Z 707.406,A -85,B 0,C 180,E1 -13175.346,E2 -13175.346} C_VEL
LIN {X 0,Y 361.863,Z 707.405,A -85,B 0,C 180,E1 -13179.028,E2 -13179.028} C_VEL
LIN {X 0,Y 361.9,Z 707.59,A -85,B 0,C 180,E1 -13182.82,E2 -13182.82} C_VEL
LIN {X 0,Y 362.168,Z 708.709,A -85,B 0,C 180,E1 -13183.018,E2 -13183.018} C_VEL
LIN {X 0,Y 370.66,Z 727.89,A -85,B 0,C 180,E1 -13184.047,E2 -13184.047} C_VEL
LIN {X 0,Y 371.222,Z 729.247,A -85,B 0,C 180,E1 -13184.113,E2 -13184.113} C_VEL
LIN {X 0,Y 370.514,Z 786.349,A -85,B 0,C 180,E1 -13185.284,E2 -13185.284} C_VEL
LIN {X 0,Y 370.377,Z 800.012,A -85,B 0,C 180,E1 -13185.718,E2 -13185.718} C_VEL
LIN {X 0,Y 370.164,Z 812.019,A -85,B 0,C 180,E1 -13186.318,E2 -13186.318} C_VEL
LIN {X 0,Y 369.614,Z 823.333,A -85,B 0,C 180,E1 -13187.08,E2 -13187.08} C_VEL
LIN {X 0,Y 368.859,Z 833.915,A -85,B 0,C 180,E1 -13187.995,E2 -13187.995} C_VEL
LIN {X 0,Y 368.007,Z 844.515,A -85,B 0,C 180,E1 -13189.152,E2 -13189.152} C_VEL
LIN {X 0,Y 367.011,Z 854.565,A -85,B 0,C 180,E1 -13190.514,E2 -13190.514} C_VEL
LIN {X 0,Y 365.953,Z 863.774,A -85,B 0,C 180,E1 -13192.083,E2 -13192.083} C_VEL
LIN {X 0,Y 364.981,Z 871.609,A -85,B 0,C 180,E1 -13193.748,E2 -13193.748} C_VEL
LIN {X 0,Y 364.265,Z 877.491,A -85,B 0,C 180,E1 -13195.311,E2 -13195.311} C_VEL
LIN {X 0,Y 363.446,Z 883.15,A -85,B 0,C 180,E1 -13197.221,E2 -13197.221} C_VEL
LIN {X 0,Y 362.918,Z 887.288,A -85,B 0,C 180,E1 -13199.126,E2 -13199.126} C_VEL
LIN {X 0,Y 362.496,Z 890.117,A -85,B 0,C 180,E1 -13201.01,E2 -13201.01} C_VEL
LIN {X 0,Y 362.309,Z 891.358,A -85,B 0,C 180,E1 -13202.256,E2 -13202.256} C_VEL
LIN {X 0,Y 362.179,Z 892.051,A -85,B 0,C 180,E1 -13203.495,E2 -13203.495} C_VEL
LIN {X 0,Y 362.078,Z 892.299,A -85,B 0,C 180,E1 -13204.723,E2 -13204.723} C_VEL
LIN {X 0,Y 362.027,Z 892.072,A -85,B 0,C 180,E1 -13205.943,E2 -13205.943} C_VEL
LIN {X 0,Y 362.078,Z 891.355,A -85,B 0,C 180,E1 -13207.159,E2 -13207.159} C_VEL
LIN {X 0,Y 362.268,Z 889.889,A -85,B 0,C 180,E1 -13208.624,E2 -13208.624} C_VEL
LIN {X 0,Y 362.669,Z 886.436,A -85,B 0,C 180,E1 -13210.767,E2 -13210.767} C_VEL
LIN {X 0,Y 363.125,Z 882.334,A -85,B 0,C 180,E1 -13212.545,E2 -13212.545} C_VEL
LIN {X 0,Y 363.733,Z 877.003,A -85,B 0,C 180,E1 -13214.307,E2 -13214.307} C_VEL
LIN {X 0,Y 364.431,Z 870.256,A -85,B 0,C 180,E1 -13216.053,E2 -13216.053} C_VEL
LIN {X 0,Y 365.383,Z 861.799,A -85,B 0,C 180,E1 -13217.787,E2 -13217.787} C_VEL
LIN {X 0,Y 366.194,Z 853.193,A -85,B 0,C 180,E1 -13219.217,E2 -13219.217} C_VEL
LIN {X 0,Y 367.035,Z 843.701,A -85,B 0,C 180,E1 -13220.496,E2 -13220.496} C_VEL
LIN {X 0,Y 367.919,Z 831.928,A -85,B 0,C 180,E1 -13221.765,E2 -13221.765} C_VEL
LIN {X 0,Y 368.654,Z 820.396,A -85,B 0,C 180,E1 -13222.736,E2 -13222.736} C_VEL
LIN {X 0,Y 369.088,Z 808.482,A -85,B 0,C 180,E1 -13223.503,E2 -13223.503} C_VEL
LIN {X 0,Y 369.395,Z 794.816,A -85,B 0,C 180,E1 -13224.128,E2 -13224.128} C_VEL
LIN {X 0,Y 369.498,Z 780.946,A -85,B 0,C 180,E1 -13224.507,E2 -13224.507} C_VEL
LIN {X 0,Y 370.12,Z 727.684,A -85,B 0,C 180,E1 -13225.573,E2 -13225.573} C_VEL
LIN {X 0,Y 362.179,Z 708.284,A -85,B 0,C 180,E1 -13226.476,E2 -13226.476} C_VEL
LIN {X 0,Y 362.043,Z 707.459,A -85,B 0,C 180,E1 -13226.698,E2 -13226.698} C_VEL
LIN {X 0,Y 362.266,Z 707.359,A -85,B 0,C 180,E1 -13227.778,E2 -13227.778} C_VEL
LIN {X 0,Y 362.177,Z 707.371,A -85,B 0,C 180,E1 -13231.114,E2 -13231.114} C_VEL
LIN {X 0,Y 362.261,Z 707.359,A -85,B 0,C 180,E1 -13232.225,E2 -13232.225} C_VEL
LIN {X 0,Y 362.123,Z 707.374,A -85,B 0,C 180,E1 -13236.689,E2 -13236.689} C_VEL
LIN {X 0,Y 361.998,Z 707.39,A -85,B 0,C 180,E1 -13240.065,E2 -13240.065} C_VEL
LIN {X 0,Y 362.004,Z 707.389,A -85,B 0,C 180,E1 -13243.9,E2 -13243.9} C_VEL
LIN {X 0,Y 361.914,Z 707.401,A -85,B 0,C 180,E1 -13247.525,E2 -13247.525} C_VEL
LIN {X 0,Y 361.252,Z 707.484,A -85,B 0,C 180,E1 -13248.454,E2 -13248.454} C_VEL
LIN {X 0,Y 358.386,Z 707.839,A -85,B 0,C 180,E1 -13249.963,E2 -13249.963} C_VEL
LIN {X 0,Y 355.945,Z 708.143,A -85,B 0,C 180,E1 -13251.184,E2 -13251.184} C_VEL
LIN {X 0,Y 354.886,Z 708.275,A -85,B 0,C 180,E1 -13252.129,E2 -13252.129} C_VEL
LIN {X 0,Y 354.794,Z 708.285,A -85,B 0,C 180,E1 -13252.45,E2 -13252.45} C_VEL
LIN {X 0,Y 354.807,Z 708.272,A -85,B 0,C 180,E1 -13255.836,E2 -13255.836} C_VEL
LIN {X 0,Y 354.799,Z 708.289,A -85,B 0,C 180,E1 -13259.685,E2 -13259.685} C_VEL
LIN {X 0,Y 354.814,Z 708.266,A -85,B 0,C 180,E1 -13263.703,E2 -13263.703} C_VEL
LIN {X 0,Y 354.798,Z 708.273,A -85,B 0,C 180,E1 -13266.461,E2 -13266.461} C_VEL
LIN {X 0,Y 354.775,Z 708.294,A -85,B 0,C 180,E1 -13269.413,E2 -13269.413} C_VEL
LIN {X 0,Y 354.773,Z 708.291,A -85,B 0,C 180,E1 -13272.864,E2 -13272.864} C_VEL
LIN {X 0,Y 354.765,Z 708.294,A -85,B 0,C 180,E1 -13276.103,E2 -13276.103} C_VEL
LIN {X 0,Y 354.769,Z 708.292,A -85,B 0,C 180,E1 -13279.176,E2 -13279.176} C_VEL
LIN {X 0,Y 354.804,Z 708.289,A -85,B 0,C 180,E1 -13282.406,E2 -13282.406} C_VEL
LIN {X 0,Y 354.897,Z 708.502,A -85,B 0,C 180,E1 -13286.06,E2 -13286.06} C_VEL
LIN {X 0,Y 355.106,Z 709.467,A -85,B 0,C 180,E1 -13286.228,E2 -13286.228} C_VEL
LIN {X 0,Y 361.598,Z 727.703,A -85,B 0,C 180,E1 -13287.002,E2 -13287.002} C_VEL
LIN {X 0,Y 360.491,Z 785.987,A -85,B 0,C 180,E1 -13288.414,E2 -13288.414} C_VEL
LIN {X 0,Y 360.299,Z 797.168,A -85,B 0,C 180,E1 -13288.85,E2 -13288.85} C_VEL
LIN {X 0,Y 360.018,Z 807.554,A -85,B 0,C 180,E1 -13289.404,E2 -13289.404} C_VEL
LIN {X 0,Y 359.569,Z 817.808,A -85,B 0,C 180,E1 -13290.105,E2 -13290.105} C_VEL
LIN {X 0,Y 359.045,Z 826.866,A -85,B 0,C 180,E1 -13290.862,E2 -13290.862} C_VEL
LIN {X 0,Y 358.546,Z 835.902,A -85,B 0,C 180,E1 -13291.778,E2 -13291.778} C_VEL
LIN {X 0,Y 357.884,Z 844.64,A -85,B 0,C 180,E1 -13292.833,E2 -13292.833} C_VEL
LIN {X 0,Y 357.343,Z 853.025,A -85,B 0,C 180,E1 -13294.049,E2 -13294.049} C_VEL
LIN {X 0,Y 356.854,Z 859.967,A -85,B 0,C 180,E1 -13295.231,E2 -13295.231} C_VEL
LIN {X 0,Y 356.206,Z 867.433,A -85,B 0,C 180,E1 -13296.758,E2 -13296.758} C_VEL
LIN {X 0,Y 355.787,Z 873.238,A -85,B 0,C 180,E1 -13298.192,E2 -13298.192} C_VEL
LIN {X 0,Y 355.41,Z 878.426,A -85,B 0,C 180,E1 -13299.754,E2 -13299.754} C_VEL
LIN {X 0,Y 355.222,Z 881.764,A -85,B 0,C 180,E1 -13300.946,E2 -13300.946} C_VEL
LIN {X 0,Y 354.982,Z 885.589,A -85,B 0,C 180,E1 -13302.724,E2 -13302.724} C_VEL
LIN {X 0,Y 354.842,Z 887.479,A -85,B 0,C 180,E1 -13303.902,E2 -13303.902} C_VEL
LIN {X 0,Y 354.853,Z 889.952,A -85,B 0,C 180,E1 -13306.251,E2 -13306.251} C_VEL
LIN {X 0,Y 354.889,Z 890.506,A -85,B 0,C 180,E1 -13307.418,E2 -13307.418} C_VEL
LIN {X 0,Y 355.034,Z 890.622,A -85,B 0,C 180,E1 -13308.582,E2 -13308.582} C_VEL
LIN {X 0,Y 355.423,Z 889.465,A -85,B 0,C 180,E1 -13310.898,E2 -13310.898} C_VEL
LIN {X 0,Y 355.994,Z 886.563,A -85,B 0,C 180,E1 -13313.197,E2 -13313.197} C_VEL
LIN {X 0,Y 356.602,Z 883.172,A -85,B 0,C 180,E1 -13314.912,E2 -13314.912} C_VEL
LIN {X 0,Y 357.031,Z 880.379,A -85,B 0,C 180,E1 -13316.049,E2 -13316.049} C_VEL
LIN {X 0,Y 357.915,Z 873.955,A -85,B 0,C 180,E1 -13318.031,E2 -13318.031} C_VEL
LIN {X 0,Y 358.663,Z 869.077,A -85,B 0,C 180,E1 -13319.252,E2 -13319.252} C_VEL
LIN {X 0,Y 359.684,Z 861.251,A -85,B 0,C 180,E1 -13320.839,E2 -13320.839} C_VEL
LIN {X 0,Y 360.492,Z 854.694,A -85,B 0,C 180,E1 -13321.955,E2 -13321.955} C_VEL
LIN {X 0,Y 361.429,Z 845.889,A -85,B 0,C 180,E1 -13323.205,E2 -13323.205} C_VEL
LIN {X 0,Y 362.245,Z 837.695,A -85,B 0,C 180,E1 -13324.172,E2 -13324.172} C_VEL
LIN {X 0,Y 363.038,Z 827.765,A -85,B 0,C 180,E1 -13325.137,E2 -13325.137} C_VEL
LIN {X 0,Y 363.587,Z 818.222,A -85,B 0,C 180,E1 -13325.894,E2 -13325.894} C_VEL
LIN {X 0,Y 364.076,Z 807.74,A -85,B 0,C 180,E1 -13326.547,E2 -13326.547} C_VEL
LIN {X 0,Y 364.413,Z 797.514,A -85,B 0,C 180,E1 -13327.027,E2 -13327.027} C_VEL
LIN {X 0,Y 364.577,Z 785.156,A -85,B 0,C 180,E1 -13327.442,E2 -13327.442} C_VEL
LIN {X 0,Y 365.188,Z 762.504,A -85,B 0,C 180,E1 -13328.039,E2 -13328.039} C_VEL
LIN {X 0,Y 366.412,Z 731.6,A -85,B 0,C 180,E1 -13328.849,E2 -13328.849} C_VEL
LIN {X 0,Y 361.187,Z 720.691,A -85,B 0,C 180,E1 -13329.69,E2 -13329.69} C_VEL
LIN {X 0,Y 356.37,Z 711.755,A -85,B 0,C 180,E1 -13330.487,E2 -13330.487} C_VEL
LIN {X 0,Y 355.068,Z 709.02,A -85,B 0,C 180,E1 -13330.766,E2 -13330.766} C_VEL
LIN {X 0,Y 354.942,Z 708.36,A -85,B 0,C 180,E1 -13330.986,E2 -13330.986} C_VEL
LIN {X 0,Y 354.951,Z 708.268,A -85,B 0,C 180,E1 -13334.018,E2 -13334.018} C_VEL
LIN {X 0,Y 354.898,Z 708.279,A -85,B 0,C 180,E1 -13338.092,E2 -13338.092} C_VEL
LIN {X 0,Y 354.826,Z 708.286,A -85,B 0,C 180,E1 -13341.417,E2 -13341.417} C_VEL
LIN {X 0,Y 354.861,Z 708.283,A -85,B 0,C 180,E1 -13344.576,E2 -13344.576} C_VEL
LIN {X 0,Y 354.817,Z 708.288,A -85,B 0,C 180,E1 -13348.384,E2 -13348.384} C_VEL
LIN {X 0,Y 354.794,Z 708.289,A -85,B 0,C 180,E1 -13352.333,E2 -13352.333} C_VEL
LIN {X 0,Y 354.829,Z 708.286,A -85,B 0,C 180,E1 -13355.698,E2 -13355.698} C_VEL
LIN {X 0,Y 354.831,Z 708.286,A -85,B 0,C 180,E1 -13359.423,E2 -13359.423} C_VEL
LIN {X 0,Y 354.795,Z 708.289,A -85,B 0,C 180,E1 -13362.866,E2 -13362.866} C_VEL
LIN {X 0,Y 354.773,Z 708.293,A -85,B 0,C 180,E1 -13366.103,E2 -13366.103} C_VEL
LIN {X 0,Y 354.794,Z 708.29,A -85,B 0,C 180,E1 -13369.178,E2 -13369.178} C_VEL
LIN {X 0,Y 354.812,Z 708.286,A -85,B 0,C 180,E1 -13372.402,E2 -13372.402} C_VEL
LIN {X 0,Y 354.862,Z 708.478,A -85,B 0,C 180,E1 -13374.184,E2 -13374.184} C_VEL
LIN {X 0,Y 358.178,Z 722.164,A -85,B 0,C 180,E1 -13377.154,E2 -13377.154} C_VEL
LIN {X 0,Y 361.143,Z 735.739,A -85,B 0,C 180,E1 -13379.925,E2 -13379.925} C_VEL
LIN {X 0,Y 361.186,Z 739.187,A -85,B 0,C 180,E1 -13380.571,E2 -13380.571} C_VEL
LIN {X 0,Y 358.813,Z 762.802,A -85,B 0,C 180,E1 -13384.784,E2 -13384.784} C_VEL
LIN {X 0,Y 358.04,Z 771.689,A -85,B 0,C 180,E1 -13386.311,E2 -13386.311} C_VEL
